        end
        sync()
      end
      $ 1628 "Direction: Base Z-"
      global move_thread_flag_1628=0
      thread move_thread_1628():
        enter_critical
        move_thread_flag_1628 = 1
        local towardsPos=calculate_point_to_move_towards(p[0.0,0.0,0.0,0.0,0.0,0.0], [0.0,0.0,-1.0], 1000.0)
        movel(towardsPos, a=0.007, v=0.007)
        move_thread_flag_1628 = 2
        exit_critical
      end
      move_thread_flag_1628 = 0
      move_thread_han_1628 = run move_thread_1628()
      while (True):
        local targetTcpDirection=get_target_tcp_speed()
        local stepsToRetract=tool_contact(direction=targetTcpDirection)
        if (stepsToRetract > 0):
          kill move_thread_han_1628
          stopl(0.02)
          local backTrackMovement=get_actual_joint_positions_history(stepsToRetract)
          local contactPose=get_forward_kin(backTrackMovement)
          local posDir=[targetTcpDirection[0],targetTcpDirection[1],targetTcpDirection[2]]
          local retractTo=contactPose
          if (norm(posDir) > 1e-6):
            local normalizedPosDir=normalize(posDir)
            local additionalRetraction=p[normalizedPosDir[0] * 0.0, normalizedPosDir[1] * 0.0, normalizedPosDir[2] * 0.0, 0, 0, 0]
            retractTo = pose_sub(contactPose, additionalRetraction)
          end
          movel(retractTo, a=0.02, v=0.1)
          $ 1629 "Until (tool_contact_detection)"
          break
        end
        sync()
      end
      $ 1630 "Popup: punto contacto alanzdo"
      popup("punto contacto alanzdo", "Mensaje", False, False, blocking=True)
      $ 1631 "Direction: Base Z+"
      global move_thread_flag_1631=0
      thread move_thread_1631():
        enter_critical
        move_thread_flag_1631 = 1
        local towardsPos=calculate_point_to_move_towards(p[0.0,0.0,0.0,0.0,0.0,0.0], [0.0,0.0,1.0], 0.002)
        movel(towardsPos, a=0.005, v=0.003)
        move_thread_flag_1631 = 2
        exit_critical
      end
      move_thread_flag_1631 = 0
      move_thread_han_1631 = run move_thread_1631()
      while (True):
        sleep(1.0E-10)
        if (move_thread_flag_1631 > 1):
          join move_thread_han_1631
          $ 1632 "Until (distance)"
          break
        end
        sync()
      end
      $ 1633 "Wait: 0.3"
      sleep(0.3)
      $ 1634 "Set CO[1]=Encender"
      set_configurable_digital_out(1, True)
      $ 1635 "Wait: 0.3"
      sleep(0.3)
      $ 1636 "Loop 1 times"
      Loop_129 = 0
      while (Loop_129 < 1):
        $ 1637 "bajar≔pose_add(get_actual_tcp_pose(), bajada_broca)"
        global bajar= pose_add ( get_actual_tcp_pose (), bajada_broca)
        $ 1638 "bajar" "breakAfter"
        movel(bajar, a=0.004, v=0.004)
        $ 1639 "subir≔pose_sub(get_actual_tcp_pose(), bajada_broca)"
        global subir= pose_sub ( get_actual_tcp_pose (), bajada_broca)
        $ 1640 "Direction: Base Z+"
        global move_thread_flag_1640=0
        thread move_thread_1640():
          enter_critical
          move_thread_flag_1640 = 1
          local towardsPos=calculate_point_to_move_towards(p[0.0,0.0,0.0,0.0,0.0,0.0], [0.0,0.0,1.0], 0.002)
          movel(towardsPos, a=0.015, v=0.015)
          move_thread_flag_1640 = 2
          exit_critical
        end
        move_thread_flag_1640 = 0
        move_thread_han_1640 = run move_thread_1640()
        while (True):
          sleep(1.0E-10)
          if (move_thread_flag_1640 > 1):
            join move_thread_han_1640
            $ 1641 "Until (distance)"
            break
          end
          sync()
        end
        $ 1642 "Set CO[1]=Apagar"
        set_configurable_digital_out(1, False)
        $ 1643 "subir" "breakAfter"
        movel(subir, a=0.015, v=0.015)
        $ 1644 "bajada_broca≔pose_sub(bajada_broca, bajada)"
        global bajada_broca= pose_sub (bajada_broca, bajada)
        Loop_129 = Loop_129 + 1
      end
      $ 1645 "Direction: Base Z+"
      global move_thread_flag_1645=0
      thread move_thread_1645():
        enter_critical
        move_thread_flag_1645 = 1
        local towardsPos=calculate_point_to_move_towards(p[0.0,0.0,0.0,0.0,0.0,0.0], [0.0,0.0,1.0], 0.08)
        movel(towardsPos, a=0.15, v=0.1)
        move_thread_flag_1645 = 2
        exit_critical
      end
      move_thread_flag_1645 = 0
      move_thread_han_1645 = run move_thread_1645()
      while (True):
        sleep(1.0E-10)
        if (move_thread_flag_1645 > 1):
          join move_thread_han_1645
          $ 1646 "Until (distance)"
          break
        end
        sync()
      end
      $ 1647 "Set CO[1]=Apagar"
      set_configurable_digital_out(1, False)
      $ 1648 "barreno_actual≔barreno_actual+1"
      global barreno_actual=barreno_actual+1
    end
    $ 1651 "Popup: Linea13 con chica Terminada!"
    popup("Linea13 con chica Terminada!", "Mensaje", False, False, blocking=True)
    $ 1652 "Linea14"
    $ 1653 "Marcar_puntos"
    $ 1654 "MoveL"
    $ 1655 "Linea14_A" "breakAfter"
    movel(Linea14_A_p, a=0.5, v=0.1)
    $ 1656 "bajada_comprobacion"
    $ 1657 "Direction: Base Z-"
    global move_thread_flag_1657=0
    thread move_thread_1657():
      enter_critical
      move_thread_flag_1657 = 1
      local towardsPos=calculate_point_to_move_towards(p[0.0,0.0,0.0,0.0,0.0,0.0], [0.0,0.0,-1.0], 0.071)
      movel(towardsPos, a=0.15, v=0.1)
      move_thread_flag_1657 = 2
      exit_critical
    end
    move_thread_flag_1657 = 0
    move_thread_han_1657 = run move_thread_1657()
    while (True):
      sleep(1.0E-10)
      if (move_thread_flag_1657 > 1):
        join move_thread_han_1657
        $ 1658 "Until (distance)"
        break
      end
      sync()
    end
    $ 1659 "Direction: Base Z-"
    global move_thread_flag_1659=0
    thread move_thread_1659():
      enter_critical
      move_thread_flag_1659 = 1
      local towardsPos=calculate_point_to_move_towards(p[0.0,0.0,0.0,0.0,0.0,0.0], [0.0,0.0,-1.0], 1000.0)
      movel(towardsPos, a=0.007, v=0.007)
      move_thread_flag_1659 = 2
      exit_critical
    end
    move_thread_flag_1659 = 0
    move_thread_han_1659 = run move_thread_1659()
    while (True):
      local targetTcpDirection=get_target_tcp_speed()
      local stepsToRetract=tool_contact(direction=targetTcpDirection)
      if (stepsToRetract > 0):
        kill move_thread_han_1659
        stopl(0.02)
        local backTrackMovement=get_actual_joint_positions_history(stepsToRetract)
        local contactPose=get_forward_kin(backTrackMovement)
        local posDir=[targetTcpDirection[0],targetTcpDirection[1],targetTcpDirection[2]]
        local retractTo=contactPose
        if (norm(posDir) > 1e-6):
          local normalizedPosDir=normalize(posDir)
          local additionalRetraction=p[normalizedPosDir[0] * 0.0, normalizedPosDir[1] * 0.0, normalizedPosDir[2] * 0.0, 0, 0, 0]
          retractTo = pose_sub(contactPose, additionalRetraction)
        end
        movel(retractTo, a=0.02, v=0.1)
        $ 1660 "Until (tool_contact_detection)"
        break
      end
      sync()
    end
    $ 1661 "Direction: Base Z+"
    global move_thread_flag_1661=0
    thread move_thread_1661():
      enter_critical
      move_thread_flag_1661 = 1
      local towardsPos=calculate_point_to_move_towards(p[0.0,0.0,0.0,0.0,0.0,0.0], [0.0,0.0,1.0], 0.08)
      movel(towardsPos, a=0.15, v=0.1)
      move_thread_flag_1661 = 2
      exit_critical
    end
    move_thread_flag_1661 = 0
    move_thread_han_1661 = run move_thread_1661()
    while (True):
      sleep(1.0E-10)
      if (move_thread_flag_1661 > 1):
        join move_thread_han_1661
        $ 1662 "Until (distance)"
        break
      end
      sync()
    end
    $ 1663 "Linea14_B" "breakAfter"
    movel(Linea14_B_p, a=0.5, v=0.1)
    $ 1664 "bajada_comprobacion"
    $ 1665 "Direction: Base Z-"
    global move_thread_flag_1665=0
    thread move_thread_1665():
      enter_critical
      move_thread_flag_1665 = 1
      local towardsPos=calculate_point_to_move_towards(p[0.0,0.0,0.0,0.0,0.0,0.0], [0.0,0.0,-1.0], 0.071)
      movel(towardsPos, a=0.15, v=0.1)
      move_thread_flag_1665 = 2
      exit_critical
    end
    move_thread_flag_1665 = 0
    move_thread_han_1665 = run move_thread_1665()
    while (True):
      sleep(1.0E-10)
      if (move_thread_flag_1665 > 1):
        join move_thread_han_1665
        $ 1666 "Until (distance)"
        break
      end
      sync()
    end
    $ 1667 "Direction: Base Z-"
    global move_thread_flag_1667=0
    thread move_thread_1667():
      enter_critical
      move_thread_flag_1667 = 1
      local towardsPos=calculate_point_to_move_towards(p[0.0,0.0,0.0,0.0,0.0,0.0], [0.0,0.0,-1.0], 1000.0)
      movel(towardsPos, a=0.007, v=0.007)
      move_thread_flag_1667 = 2
      exit_critical
    end
    move_thread_flag_1667 = 0
    move_thread_han_1667 = run move_thread_1667()
    while (True):
      local targetTcpDirection=get_target_tcp_speed()
      local stepsToRetract=tool_contact(direction=targetTcpDirection)
      if (stepsToRetract > 0):
        kill move_thread_han_1667
        stopl(0.02)
        local backTrackMovement=get_actual_joint_positions_history(stepsToRetract)
        local contactPose=get_forward_kin(backTrackMovement)
        local posDir=[targetTcpDirection[0],targetTcpDirection[1],targetTcpDirection[2]]
        local retractTo=contactPose
        if (norm(posDir) > 1e-6):
          local normalizedPosDir=normalize(posDir)
          local additionalRetraction=p[normalizedPosDir[0] * 0.0, normalizedPosDir[1] * 0.0, normalizedPosDir[2] * 0.0, 0, 0, 0]
          retractTo = pose_sub(contactPose, additionalRetraction)
        end
        movel(retractTo, a=0.02, v=0.1)
        $ 1668 "Until (tool_contact_detection)"
        break
      end
      sync()
    end
    $ 1669 "Direction: Base Z+"
    global move_thread_flag_1669=0
    thread move_thread_1669():
      enter_critical
      move_thread_flag_1669 = 1
      local towardsPos=calculate_point_to_move_towards(p[0.0,0.0,0.0,0.0,0.0,0.0], [0.0,0.0,1.0], 0.08)
      movel(towardsPos, a=0.15, v=0.1)
      move_thread_flag_1669 = 2
      exit_critical
    end
    move_thread_flag_1669 = 0
    move_thread_han_1669 = run move_thread_1669()
    while (True):
      sleep(1.0E-10)
      if (move_thread_flag_1669 > 1):
        join move_thread_han_1669
        $ 1670 "Until (distance)"
        break
      end
      sync()
    end
    $ 1671 "AB"
    $ 1672 "'desbaste_inicial'"
    # 'desbaste_inicial'
    $ 1673 "bajada_broca≔p[0,0,-0.008,0,0,0]"
    global bajada_broca=p[0,0,-0.008,0,0,0]
    $ 1674 "barrenos_menos1≔5"
    global barrenos_menos1=5
    $ 1675 "barreno_actual≔0"
    global barreno_actual=0
    $ 1676 "Loop barreno_actual≤barrenos_menos1"
    while (barreno_actual <= barrenos_menos1):
      $ 1677 "Perforacion"
      $ 1678 "MoveL"
      $ 1679 "If barreno_actual≟3"
      if (barreno_actual == 3):
        $ 1680 "barreno_actual≔barreno_actual+1"
        global barreno_actual=barreno_actual+1
      end
      $ 1681 "internos≔interpolate_pose(Linea14_A, Linea14_B, barreno_actual/barrenos_menos1)"
      global internos= interpolate_pose (Linea14_A_p, Linea14_B_p, barreno_actual/barrenos_menos1)
      $ 1682 "internos" "breakAfter"
      movel(internos, a=0.5, v=0.1)
      $ 1683 "'desbaste_inicial'"
      # 'desbaste_inicial'
      $ 1684 "bajada_broca≔p[0,0,-0.024,0,0,0]"
      global bajada_broca=p[0,0,-0.024,0,0,0]
      $ 1685 "bajada≔p[0,0,0.024,0,0,0]"
      global bajada=p[0,0,0.024,0,0,0]
      $ 1686 "Direction: Base Z-"
      global move_thread_flag_1686=0
      thread move_thread_1686():
        enter_critical
        move_thread_flag_1686 = 1
        local towardsPos=calculate_point_to_move_towards(p[0.0,0.0,0.0,0.0,0.0,0.0], [0.0,0.0,-1.0], 0.071)
        movel(towardsPos, a=0.15, v=0.1)
        move_thread_flag_1686 = 2
        exit_critical
      end
      move_thread_flag_1686 = 0
      move_thread_han_1686 = run move_thread_1686()
      while (True):
        sleep(1.0E-10)
        if (move_thread_flag_1686 > 1):
          join move_thread_han_1686
          $ 1687 "Until (distance)"
          break
        end
        sync()
      end
      $ 1688 "Direction: Base Z-"
      global move_thread_flag_1688=0
      thread move_thread_1688():
        enter_critical
        move_thread_flag_1688 = 1
        local towardsPos=calculate_point_to_move_towards(p[0.0,0.0,0.0,0.0,0.0,0.0], [0.0,0.0,-1.0], 1000.0)
        movel(towardsPos, a=0.007, v=0.007)
        move_thread_flag_1688 = 2
        exit_critical
      end
      move_thread_flag_1688 = 0
      move_thread_han_1688 = run move_thread_1688()
      while (True):
        local targetTcpDirection=get_target_tcp_speed()
        local stepsToRetract=tool_contact(direction=targetTcpDirection)
        if (stepsToRetract > 0):
          kill move_thread_han_1688
          stopl(0.02)
          local backTrackMovement=get_actual_joint_positions_history(stepsToRetract)
          local contactPose=get_forward_kin(backTrackMovement)
          local posDir=[targetTcpDirection[0],targetTcpDirection[1],targetTcpDirection[2]]
          local retractTo=contactPose
          if (norm(posDir) > 1e-6):
            local normalizedPosDir=normalize(posDir)
            local additionalRetraction=p[normalizedPosDir[0] * 0.0, normalizedPosDir[1] * 0.0, normalizedPosDir[2] * 0.0, 0, 0, 0]
            retractTo = pose_sub(contactPose, additionalRetraction)
          end
          movel(retractTo, a=0.02, v=0.1)
          $ 1689 "Until (tool_contact_detection)"
          break
        end
        sync()
      end
      $ 1690 "Popup: punto contacto alanzdo"
      popup("punto contacto alanzdo", "Mensaje", False, False, blocking=True)
      $ 1691 "Direction: Base Z+"
      global move_thread_flag_1691=0
      thread move_thread_1691():
        enter_critical
        move_thread_flag_1691 = 1
        local towardsPos=calculate_point_to_move_towards(p[0.0,0.0,0.0,0.0,0.0,0.0], [0.0,0.0,1.0], 0.002)
        movel(towardsPos, a=0.005, v=0.003)
        move_thread_flag_1691 = 2
        exit_critical
      end
      move_thread_flag_1691 = 0
      move_thread_han_1691 = run move_thread_1691()
      while (True):
        sleep(1.0E-10)
        if (move_thread_flag_1691 > 1):
          join move_thread_han_1691
          $ 1692 "Until (distance)"
          break
        end
        sync()
      end
      $ 1693 "Wait: 0.3"
      sleep(0.3)
      $ 1694 "Set CO[1]=Encender"
      set_configurable_digital_out(1, True)
      $ 1695 "Wait: 0.3"
      sleep(0.3)
      $ 1696 "Loop 1 times"
      Loop_131 = 0
      while (Loop_131 < 1):
        $ 1697 "bajar≔pose_add(get_actual_tcp_pose(), bajada_broca)"
        global bajar= pose_add ( get_actual_tcp_pose (), bajada_broca)
        $ 1698 "bajar" "breakAfter"
        movel(bajar, a=0.004, v=0.004)
        $ 1699 "subir≔pose_sub(get_actual_tcp_pose(), bajada_broca)"
        global subir= pose_sub ( get_actual_tcp_pose (), bajada_broca)
        $ 1700 "Direction: Base Z+"
        global move_thread_flag_1700=0
        thread move_thread_1700():
          enter_critical
          move_thread_flag_1700 = 1
          local towardsPos=calculate_point_to_move_towards(p[0.0,0.0,0.0,0.0,0.0,0.0], [0.0,0.0,1.0], 0.002)
          movel(towardsPos, a=0.015, v=0.015)
          move_thread_flag_1700 = 2
          exit_critical
        end
        move_thread_flag_1700 = 0
        move_thread_han_1700 = run move_thread_1700()
        while (True):
          sleep(1.0E-10)
          if (move_thread_flag_1700 > 1):
            join move_thread_han_1700
            $ 1701 "Until (distance)"
            break
          end
          sync()
        end
        $ 1702 "Set CO[1]=Apagar"
        set_configurable_digital_out(1, False)
        $ 1703 "subir" "breakAfter"
        movel(subir, a=0.015, v=0.015)
        $ 1704 "bajada_broca≔pose_sub(bajada_broca, bajada)"
        global bajada_broca= pose_sub (bajada_broca, bajada)
        Loop_131 = Loop_131 + 1
      end
      $ 1705 "Direction: Base Z+"
      global move_thread_flag_1705=0
      thread move_thread_1705():
        enter_critical
        move_thread_flag_1705 = 1
        local towardsPos=calculate_point_to_move_towards(p[0.0,0.0,0.0,0.0,0.0,0.0], [0.0,0.0,1.0], 0.08)
        movel(towardsPos, a=0.15, v=0.1)
        move_thread_flag_1705 = 2
        exit_critical
      end
      move_thread_flag_1705 = 0
      move_thread_han_1705 = run move_thread_1705()
      while (True):
        sleep(1.0E-10)
        if (move_thread_flag_1705 > 1):
          join move_thread_han_1705
          $ 1706 "Until (distance)"
          break
        end
        sync()
      end
      $ 1707 "Set CO[1]=Apagar"
      set_configurable_digital_out(1, False)
      $ 1708 "barreno_actual≔barreno_actual+1"
      global barreno_actual=barreno_actual+1
    end
    $ 1711 "Popup: Linea14 con chica Terminada!"
    popup("Linea14 con chica Terminada!", "Mensaje", False, False, blocking=True)
    $ 1712 "Linea15"
    $ 1713 "Marcar_puntos"
    $ 1714 "MoveL"
    $ 1715 "Linea15_A" "breakAfter"
    movel(Linea15_A_p, a=0.5, v=0.1)
    $ 1716 "bajada_comprobacion"
    $ 1717 "Direction: Base Z-"
    global move_thread_flag_1717=0
    thread move_thread_1717():
      enter_critical
      move_thread_flag_1717 = 1
      local towardsPos=calculate_point_to_move_towards(p[0.0,0.0,0.0,0.0,0.0,0.0], [0.0,0.0,-1.0], 0.071)
      movel(towardsPos, a=0.15, v=0.1)
      move_thread_flag_1717 = 2
      exit_critical
    end
    move_thread_flag_1717 = 0
    move_thread_han_1717 = run move_thread_1717()
    while (True):
      sleep(1.0E-10)
      if (move_thread_flag_1717 > 1):
        join move_thread_han_1717
        $ 1718 "Until (distance)"
        break
      end
      sync()
    end
    $ 1719 "Direction: Base Z-"
    global move_thread_flag_1719=0
    thread move_thread_1719():
      enter_critical
      move_thread_flag_1719 = 1
      local towardsPos=calculate_point_to_move_towards(p[0.0,0.0,0.0,0.0,0.0,0.0], [0.0,0.0,-1.0], 1000.0)
      movel(towardsPos, a=0.007, v=0.007)
      move_thread_flag_1719 = 2
      exit_critical
    end
    move_thread_flag_1719 = 0
    move_thread_han_1719 = run move_thread_1719()
    while (True):
      local targetTcpDirection=get_target_tcp_speed()
      local stepsToRetract=tool_contact(direction=targetTcpDirection)
      if (stepsToRetract > 0):
        kill move_thread_han_1719
        stopl(0.02)
        local backTrackMovement=get_actual_joint_positions_history(stepsToRetract)
        local contactPose=get_forward_kin(backTrackMovement)
        local posDir=[targetTcpDirection[0],targetTcpDirection[1],targetTcpDirection[2]]
        local retractTo=contactPose
        if (norm(posDir) > 1e-6):
          local normalizedPosDir=normalize(posDir)
          local additionalRetraction=p[normalizedPosDir[0] * 0.0, normalizedPosDir[1] * 0.0, normalizedPosDir[2] * 0.0, 0, 0, 0]
          retractTo = pose_sub(contactPose, additionalRetraction)
        end
        movel(retractTo, a=0.02, v=0.1)
        $ 1720 "Until (tool_contact_detection)"
        break
      end
      sync()
    end
    $ 1721 "Direction: Base Z+"
    global move_thread_flag_1721=0
    thread move_thread_1721():
      enter_critical
      move_thread_flag_1721 = 1
      local towardsPos=calculate_point_to_move_towards(p[0.0,0.0,0.0,0.0,0.0,0.0], [0.0,0.0,1.0], 0.08)
      movel(towardsPos, a=0.15, v=0.1)
      move_thread_flag_1721 = 2
      exit_critical
    end
    move_thread_flag_1721 = 0
    move_thread_han_1721 = run move_thread_1721()
    while (True):
      sleep(1.0E-10)
      if (move_thread_flag_1721 > 1):
        join move_thread_han_1721
        $ 1722 "Until (distance)"
        break
      end
      sync()
    end
    $ 1723 "Linea15_B" "breakAfter"
    movel(Linea15_B_p, a=0.5, v=0.1)
    $ 1724 "bajada_comprobacion"
    $ 1725 "Direction: Base Z-"
    global move_thread_flag_1725=0
    thread move_thread_1725():
      enter_critical
      move_thread_flag_1725 = 1
      local towardsPos=calculate_point_to_move_towards(p[0.0,0.0,0.0,0.0,0.0,0.0], [0.0,0.0,-1.0], 0.071)
      movel(towardsPos, a=0.15, v=0.1)
      move_thread_flag_1725 = 2
      exit_critical
    end
    move_thread_flag_1725 = 0
    move_thread_han_1725 = run move_thread_1725()
    while (True):
      sleep(1.0E-10)
      if (move_thread_flag_1725 > 1):
        join move_thread_han_1725
        $ 1726 "Until (distance)"
        break
      end
      sync()
    end
    $ 1727 "Direction: Base Z-"
    global move_thread_flag_1727=0
    thread move_thread_1727():
      enter_critical
      move_thread_flag_1727 = 1
      local towardsPos=calculate_point_to_move_towards(p[0.0,0.0,0.0,0.0,0.0,0.0], [0.0,0.0,-1.0], 1000.0)
      movel(towardsPos, a=0.007, v=0.007)
      move_thread_flag_1727 = 2
      exit_critical
    end
    move_thread_flag_1727 = 0
    move_thread_han_1727 = run move_thread_1727()
    while (True):
      local targetTcpDirection=get_target_tcp_speed()
      local stepsToRetract=tool_contact(direction=targetTcpDirection)
      if (stepsToRetract > 0):
        kill move_thread_han_1727
        stopl(0.02)
        local backTrackMovement=get_actual_joint_positions_history(stepsToRetract)
        local contactPose=get_forward_kin(backTrackMovement)
        local posDir=[targetTcpDirection[0],targetTcpDirection[1],targetTcpDirection[2]]
        local retractTo=contactPose
        if (norm(posDir) > 1e-6):
          local normalizedPosDir=normalize(posDir)
          local additionalRetraction=p[normalizedPosDir[0] * 0.0, normalizedPosDir[1] * 0.0, normalizedPosDir[2] * 0.0, 0, 0, 0]
          retractTo = pose_sub(contactPose, additionalRetraction)
        end
        movel(retractTo, a=0.02, v=0.1)
        $ 1728 "Until (tool_contact_detection)"
        break
      end
      sync()
    end
    $ 1729 "Direction: Base Z+"
    global move_thread_flag_1729=0
    thread move_thread_1729():
      enter_critical
      move_thread_flag_1729 = 1
      local towardsPos=calculate_point_to_move_towards(p[0.0,0.0,0.0,0.0,0.0,0.0], [0.0,0.0,1.0], 0.08)
      movel(towardsPos, a=0.15, v=0.1)
      move_thread_flag_1729 = 2
      exit_critical
    end
    move_thread_flag_1729 = 0
    move_thread_han_1729 = run move_thread_1729()
    while (True):
      sleep(1.0E-10)
      if (move_thread_flag_1729 > 1):
        join move_thread_han_1729
        $ 1730 "Until (distance)"
        break
      end
      sync()
    end
    $ 1731 "AB"
    $ 1732 "'desbaste_inicial'"
    # 'desbaste_inicial'
    $ 1733 "bajada_broca≔p[0,0,-0.008,0,0,0]"
    global bajada_broca=p[0,0,-0.008,0,0,0]
    $ 1734 "barrenos_menos1≔3"
    global barrenos_menos1=3
    $ 1735 "barreno_actual≔0"
    global barreno_actual=0
    $ 1736 "Loop barreno_actual≤barrenos_menos1"
    while (barreno_actual <= barrenos_menos1):
      $ 1737 "Perforacion"
      $ 1738 "MoveL"
      $ 1741 "internos≔interpolate_pose(Linea15_A, Linea15_B, barreno_actual/barrenos_menos1)"
      global internos= interpolate_pose (Linea15_A_p, Linea15_B_p, barreno_actual/barrenos_menos1)
      $ 1742 "internos" "breakAfter"
      movel(internos, a=0.5, v=0.1)
      $ 1743 "'desbaste_inicial'"
      # 'desbaste_inicial'
      $ 1744 "bajada_broca≔p[0,0,-0.024,0,0,0]"
      global bajada_broca=p[0,0,-0.024,0,0,0]
      $ 1745 "bajada≔p[0,0,0.024,0,0,0]"
      global bajada=p[0,0,0.024,0,0,0]
      $ 1746 "Direction: Base Z-"
      global move_thread_flag_1746=0
      thread move_thread_1746():
        enter_critical
        move_thread_flag_1746 = 1
        local towardsPos=calculate_point_to_move_towards(p[0.0,0.0,0.0,0.0,0.0,0.0], [0.0,0.0,-1.0], 0.071)
        movel(towardsPos, a=0.15, v=0.1)
        move_thread_flag_1746 = 2
        exit_critical
      end
      move_thread_flag_1746 = 0
      move_thread_han_1746 = run move_thread_1746()
      while (True):
        sleep(1.0E-10)
        if (move_thread_flag_1746 > 1):
          join move_thread_han_1746
          $ 1747 "Until (distance)"
          break
        end
        sync()
      end
      $ 1748 "Direction: Base Z-"
      global move_thread_flag_1748=0
      thread move_thread_1748():
        enter_critical
        move_thread_flag_1748 = 1
        local towardsPos=calculate_point_to_move_towards(p[0.0,0.0,0.0,0.0,0.0,0.0], [0.0,0.0,-1.0], 1000.0)
        movel(towardsPos, a=0.007, v=0.007)
        move_thread_flag_1748 = 2
        exit_critical
      end
      move_thread_flag_1748 = 0
      move_thread_han_1748 = run move_thread_1748()
      while (True):
        local targetTcpDirection=get_target_tcp_speed()
        local stepsToRetract=tool_contact(direction=targetTcpDirection)
        if (stepsToRetract > 0):
          kill move_thread_han_1748
          stopl(0.02)
          local backTrackMovement=get_actual_joint_positions_history(stepsToRetract)
          local contactPose=get_forward_kin(backTrackMovement)
          local posDir=[targetTcpDirection[0],targetTcpDirection[1],targetTcpDirection[2]]
          local retractTo=contactPose
          if (norm(posDir) > 1e-6):
            local normalizedPosDir=normalize(posDir)
            local additionalRetraction=p[normalizedPosDir[0] * 0.0, normalizedPosDir[1] * 0.0, normalizedPosDir[2] * 0.0, 0, 0, 0]
            retractTo = pose_sub(contactPose, additionalRetraction)
          end
          movel(retractTo, a=0.02, v=0.1)
          $ 1749 "Until (tool_contact_detection)"
          break
        end
        sync()
      end
      $ 1750 "Popup: punto contacto alanzdo"
      popup("punto contacto alanzdo", "Mensaje", False, False, blocking=True)
      $ 1751 "Direction: Base Z+"
      global move_thread_flag_1751=0
      thread move_thread_1751():
        enter_critical
        move_thread_flag_1751 = 1
        local towardsPos=calculate_point_to_move_towards(p[0.0,0.0,0.0,0.0,0.0,0.0], [0.0,0.0,1.0], 0.002)
        movel(towardsPos, a=0.005, v=0.003)
        move_thread_flag_1751 = 2
        exit_critical
      end
      move_thread_flag_1751 = 0
      move_thread_han_1751 = run move_thread_1751()
      while (True):
        sleep(1.0E-10)
        if (move_thread_flag_1751 > 1):
          join move_thread_han_1751
          $ 1752 "Until (distance)"
          break
        end
        sync()
      end
      $ 1753 "Wait: 0.3"
      sleep(0.3)
      $ 1754 "Set CO[1]=Encender"
      set_configurable_digital_out(1, True)
      $ 1755 "Wait: 0.3"
      sleep(0.3)
      $ 1756 "Loop 1 times"
      Loop_133 = 0
      while (Loop_133 < 1):
        $ 1757 "bajar≔pose_add(get_actual_tcp_pose(), bajada_broca)"
        global bajar= pose_add ( get_actual_tcp_pose (), bajada_broca)
        $ 1758 "bajar" "breakAfter"
        movel(bajar, a=0.004, v=0.004)
        $ 1759 "subir≔pose_sub(get_actual_tcp_pose(), bajada_broca)"
        global subir= pose_sub ( get_actual_tcp_pose (), bajada_broca)
        $ 1760 "Direction: Base Z+"
        global move_thread_flag_1760=0
        thread move_thread_1760():
          enter_critical
          move_thread_flag_1760 = 1
          local towardsPos=calculate_point_to_move_towards(p[0.0,0.0,0.0,0.0,0.0,0.0], [0.0,0.0,1.0], 0.002)
          movel(towardsPos, a=0.015, v=0.015)
          move_thread_flag_1760 = 2
          exit_critical
        end
        move_thread_flag_1760 = 0
        move_thread_han_1760 = run move_thread_1760()
        while (True):
          sleep(1.0E-10)
          if (move_thread_flag_1760 > 1):
            join move_thread_han_1760
            $ 1761 "Until (distance)"
            break
          end
          sync()
        end
        $ 1762 "Set CO[1]=Apagar"
        set_configurable_digital_out(1, False)
        $ 1763 "subir" "breakAfter"
        movel(subir, a=0.015, v=0.015)
        $ 1764 "bajada_broca≔pose_sub(bajada_broca, bajada)"
        global bajada_broca= pose_sub (bajada_broca, bajada)
        Loop_133 = Loop_133 + 1
      end
      $ 1765 "Direction: Base Z+"
      global move_thread_flag_1765=0
      thread move_thread_1765():
        enter_critical
        move_thread_flag_1765 = 1
        local towardsPos=calculate_point_to_move_towards(p[0.0,0.0,0.0,0.0,0.0,0.0], [0.0,0.0,1.0], 0.08)
        movel(towardsPos, a=0.15, v=0.1)
        move_thread_flag_1765 = 2
        exit_critical
      end
      move_thread_flag_1765 = 0
      move_thread_han_1765 = run move_thread_1765()
      while (True):
        sleep(1.0E-10)
        if (move_thread_flag_1765 > 1):
          join move_thread_han_1765
          $ 1766 "Until (distance)"
          break
        end
        sync()
      end
      $ 1767 "Set CO[1]=Apagar"
      set_configurable_digital_out(1, False)
      $ 1768 "barreno_actual≔barreno_actual+1"
      global barreno_actual=barreno_actual+1
    end
    $ 1771 "Popup: Linea15 con chica Terminada!"
    popup("Linea15 con chica Terminada!", "Mensaje", False, False, blocking=True)
    $ 1772 "Linea16"
    $ 1773 "Marcar_puntos"
    $ 1774 "MoveL"
    $ 1775 "Linea16_A" "breakAfter"
    movel(Linea16_A_p, a=0.5, v=0.1)
    $ 1776 "bajada_comprobacion"
    $ 1777 "Direction: Base Z-"
    global move_thread_flag_1777=0
    thread move_thread_1777():
      enter_critical
      move_thread_flag_1777 = 1
      local towardsPos=calculate_point_to_move_towards(p[0.0,0.0,0.0,0.0,0.0,0.0], [0.0,0.0,-1.0], 0.071)
      movel(towardsPos, a=0.15, v=0.1)
      move_thread_flag_1777 = 2
      exit_critical
    end
    move_thread_flag_1777 = 0
    move_thread_han_1777 = run move_thread_1777()
    while (True):
      sleep(1.0E-10)
      if (move_thread_flag_1777 > 1):
        join move_thread_han_1777
        $ 1778 "Until (distance)"
        break
      end
      sync()
    end
    $ 1779 "Direction: Base Z-"
    global move_thread_flag_1779=0
    thread move_thread_1779():
      enter_critical
      move_thread_flag_1779 = 1
      local towardsPos=calculate_point_to_move_towards(p[0.0,0.0,0.0,0.0,0.0,0.0], [0.0,0.0,-1.0], 1000.0)
      movel(towardsPos, a=0.007, v=0.007)
      move_thread_flag_1779 = 2
      exit_critical
    end
    move_thread_flag_1779 = 0
    move_thread_han_1779 = run move_thread_1779()
    while (True):
      local targetTcpDirection=get_target_tcp_speed()
      local stepsToRetract=tool_contact(direction=targetTcpDirection)
      if (stepsToRetract > 0):
        kill move_thread_han_1779
        stopl(0.02)
        local backTrackMovement=get_actual_joint_positions_history(stepsToRetract)
        local contactPose=get_forward_kin(backTrackMovement)
        local posDir=[targetTcpDirection[0],targetTcpDirection[1],targetTcpDirection[2]]
        local retractTo=contactPose
        if (norm(posDir) > 1e-6):
          local normalizedPosDir=normalize(posDir)
          local additionalRetraction=p[normalizedPosDir[0] * 0.0, normalizedPosDir[1] * 0.0, normalizedPosDir[2] * 0.0, 0, 0, 0]
          retractTo = pose_sub(contactPose, additionalRetraction)
        end
        movel(retractTo, a=0.02, v=0.1)
        $ 1780 "Until (tool_contact_detection)"
        break
      end
      sync()
    end
    $ 1781 "Direction: Base Z+"
    global move_thread_flag_1781=0
    thread move_thread_1781():
      enter_critical
      move_thread_flag_1781 = 1
      local towardsPos=calculate_point_to_move_towards(p[0.0,0.0,0.0,0.0,0.0,0.0], [0.0,0.0,1.0], 0.08)
      movel(towardsPos, a=0.15, v=0.1)
      move_thread_flag_1781 = 2
      exit_critical
    end
    move_thread_flag_1781 = 0
    move_thread_han_1781 = run move_thread_1781()
    while (True):
      sleep(1.0E-10)
      if (move_thread_flag_1781 > 1):
        join move_thread_han_1781
        $ 1782 "Until (distance)"
        break
      end
      sync()
    end
    $ 1783 "Linea16_B" "breakAfter"
    movel(Linea16_B_p, a=0.5, v=0.1)
    $ 1784 "bajada_comprobacion"
    $ 1785 "Direction: Base Z-"
    global move_thread_flag_1785=0
    thread move_thread_1785():
      enter_critical
      move_thread_flag_1785 = 1
      local towardsPos=calculate_point_to_move_towards(p[0.0,0.0,0.0,0.0,0.0,0.0], [0.0,0.0,-1.0], 0.071)
      movel(towardsPos, a=0.15, v=0.1)
      move_thread_flag_1785 = 2
      exit_critical
    end
    move_thread_flag_1785 = 0
    move_thread_han_1785 = run move_thread_1785()
    while (True):
      sleep(1.0E-10)
      if (move_thread_flag_1785 > 1):
        join move_thread_han_1785
        $ 1786 "Until (distance)"
        break
      end
      sync()
    end
    $ 1787 "Direction: Base Z-"
    global move_thread_flag_1787=0
    thread move_thread_1787():
      enter_critical
      move_thread_flag_1787 = 1
      local towardsPos=calculate_point_to_move_towards(p[0.0,0.0,0.0,0.0,0.0,0.0], [0.0,0.0,-1.0], 1000.0)
      movel(towardsPos, a=0.007, v=0.007)
      move_thread_flag_1787 = 2
      exit_critical
    end
    move_thread_flag_1787 = 0
    move_thread_han_1787 = run move_thread_1787()
    while (True):
      local targetTcpDirection=get_target_tcp_speed()
      local stepsToRetract=tool_contact(direction=targetTcpDirection)
      if (stepsToRetract > 0):
        kill move_thread_han_1787
        stopl(0.02)
        local backTrackMovement=get_actual_joint_positions_history(stepsToRetract)
        local contactPose=get_forward_kin(backTrackMovement)
        local posDir=[targetTcpDirection[0],targetTcpDirection[1],targetTcpDirection[2]]
        local retractTo=contactPose
        if (norm(posDir) > 1e-6):
          local normalizedPosDir=normalize(posDir)
          local additionalRetraction=p[normalizedPosDir[0] * 0.0, normalizedPosDir[1] * 0.0, normalizedPosDir[2] * 0.0, 0, 0, 0]
          retractTo = pose_sub(contactPose, additionalRetraction)
        end
        movel(retractTo, a=0.02, v=0.1)
        $ 1788 "Until (tool_contact_detection)"
        break
      end
      sync()
    end
    $ 1789 "Direction: Base Z+"
    global move_thread_flag_1789=0
    thread move_thread_1789():
      enter_critical
      move_thread_flag_1789 = 1
      local towardsPos=calculate_point_to_move_towards(p[0.0,0.0,0.0,0.0,0.0,0.0], [0.0,0.0,1.0], 0.08)
      movel(towardsPos, a=0.15, v=0.1)
      move_thread_flag_1789 = 2
      exit_critical
    end
    move_thread_flag_1789 = 0
    move_thread_han_1789 = run move_thread_1789()
    while (True):
      sleep(1.0E-10)
      if (move_thread_flag_1789 > 1):
        join move_thread_han_1789
        $ 1790 "Until (distance)"
        break
      end
      sync()
    end
    $ 1791 "AB"
    $ 1792 "'desbaste_inicial'"
    # 'desbaste_inicial'
    $ 1793 "bajada_broca≔p[0,0,-0.008,0,0,0]"
    global bajada_broca=p[0,0,-0.008,0,0,0]
    $ 1794 "barrenos_menos1≔1"
    global barrenos_menos1=1
    $ 1795 "barreno_actual≔0"
    global barreno_actual=0
    $ 1796 "Loop barreno_actual≤barrenos_menos1"
    while (barreno_actual <= barrenos_menos1):
      $ 1797 "Perforacion"
      $ 1798 "MoveL"
      $ 1801 "internos≔interpolate_pose(Linea16_A, Linea16_B, barreno_actual/barrenos_menos1)"
      global internos= interpolate_pose (Linea16_A_p, Linea16_B_p, barreno_actual/barrenos_menos1)
      $ 1802 "internos" "breakAfter"
      movel(internos, a=0.5, v=0.1)
      $ 1803 "'desbaste_inicial'"
      # 'desbaste_inicial'
      $ 1804 "bajada_broca≔p[0,0,-0.024,0,0,0]"
      global bajada_broca=p[0,0,-0.024,0,0,0]
      $ 1805 "bajada≔p[0,0,0.024,0,0,0]"
      global bajada=p[0,0,0.024,0,0,0]
      $ 1806 "Direction: Base Z-"
      global move_thread_flag_1806=0
      thread move_thread_1806():
        enter_critical
        move_thread_flag_1806 = 1
        local towardsPos=calculate_point_to_move_towards(p[0.0,0.0,0.0,0.0,0.0,0.0], [0.0,0.0,-1.0], 0.071)
        movel(towardsPos, a=0.15, v=0.1)
        move_thread_flag_1806 = 2
        exit_critical
      end
      move_thread_flag_1806 = 0
      move_thread_han_1806 = run move_thread_1806()
      while (True):
        sleep(1.0E-10)
        if (move_thread_flag_1806 > 1):
          join move_thread_han_1806
          $ 1807 "Until (distance)"
          break
        end
        sync()
      end
      $ 1808 "Direction: Base Z-"
      global move_thread_flag_1808=0
      thread move_thread_1808():
        enter_critical
        move_thread_flag_1808 = 1
        local towardsPos=calculate_point_to_move_towards(p[0.0,0.0,0.0,0.0,0.0,0.0], [0.0,0.0,-1.0], 1000.0)
        movel(towardsPos, a=0.007, v=0.007)
        move_thread_flag_1808 = 2
        exit_critical
      end
      move_thread_flag_1808 = 0
      move_thread_han_1808 = run move_thread_1808()
      while (True):
        local targetTcpDirection=get_target_tcp_speed()
        local stepsToRetract=tool_contact(direction=targetTcpDirection)
        if (stepsToRetract > 0):
          kill move_thread_han_1808
          stopl(0.02)
          local backTrackMovement=get_actual_joint_positions_history(stepsToRetract)
          local contactPose=get_forward_kin(backTrackMovement)
          local posDir=[targetTcpDirection[0],targetTcpDirection[1],targetTcpDirection[2]]
          local retractTo=contactPose
          if (norm(posDir) > 1e-6):
            local normalizedPosDir=normalize(posDir)
            local additionalRetraction=p[normalizedPosDir[0] * 0.0, normalizedPosDir[1] * 0.0, normalizedPosDir[2] * 0.0, 0, 0, 0]
            retractTo = pose_sub(contactPose, additionalRetraction)
          end
          movel(retractTo, a=0.02, v=0.1)
          $ 1809 "Until (tool_contact_detection)"
          break
        end
        sync()
      end
      $ 1810 "Popup: punto contacto alanzdo"
      popup("punto contacto alanzdo", "Mensaje", False, False, blocking=True)
      $ 1811 "Direction: Base Z+"
      global move_thread_flag_1811=0
      thread move_thread_1811():
        enter_critical
        move_thread_flag_1811 = 1
        local towardsPos=calculate_point_to_move_towards(p[0.0,0.0,0.0,0.0,0.0,0.0], [0.0,0.0,1.0], 0.002)
        movel(towardsPos, a=0.005, v=0.003)
        move_thread_flag_1811 = 2
        exit_critical
      end
      move_thread_flag_1811 = 0
      move_thread_han_1811 = run move_thread_1811()
      while (True):
        sleep(1.0E-10)
        if (move_thread_flag_1811 > 1):
          join move_thread_han_1811
          $ 1812 "Until (distance)"
          break
        end
        sync()
      end
      $ 1813 "Wait: 0.3"
      sleep(0.3)
      $ 1814 "Set CO[1]=Encender"
      set_configurable_digital_out(1, True)
      $ 1815 "Wait: 0.3"
      sleep(0.3)
      $ 1816 "Loop 1 times"
      Loop_135 = 0
      while (Loop_135 < 1):
        $ 1817 "bajar≔pose_add(get_actual_tcp_pose(), bajada_broca)"
        global bajar= pose_add ( get_actual_tcp_pose (), bajada_broca)
        $ 1818 "bajar" "breakAfter"
        movel(bajar, a=0.004, v=0.004)
        $ 1819 "subir≔pose_sub(get_actual_tcp_pose(), bajada_broca)"
        global subir= pose_sub ( get_actual_tcp_pose (), bajada_broca)
        $ 1820 "Direction: Base Z+"
        global move_thread_flag_1820=0
        thread move_thread_1820():
          enter_critical
          move_thread_flag_1820 = 1
          local towardsPos=calculate_point_to_move_towards(p[0.0,0.0,0.0,0.0,0.0,0.0], [0.0,0.0,1.0], 0.002)
          movel(towardsPos, a=0.015, v=0.015)
          move_thread_flag_1820 = 2
          exit_critical
        end
        move_thread_flag_1820 = 0
        move_thread_han_1820 = run move_thread_1820()
        while (True):
          sleep(1.0E-10)
          if (move_thread_flag_1820 > 1):
            join move_thread_han_1820
            $ 1821 "Until (distance)"
            break
          end
          sync()
        end
        $ 1822 "Set CO[1]=Apagar"
        set_configurable_digital_out(1, False)
        $ 1823 "subir" "breakAfter"
        movel(subir, a=0.015, v=0.015)
        $ 1824 "bajada_broca≔pose_sub(bajada_broca, bajada)"
        global bajada_broca= pose_sub (bajada_broca, bajada)
        Loop_135 = Loop_135 + 1
      end
      $ 1825 "Direction: Base Z+"
      global move_thread_flag_1825=0
      thread move_thread_1825():
        enter_critical
        move_thread_flag_1825 = 1
        local towardsPos=calculate_point_to_move_towards(p[0.0,0.0,0.0,0.0,0.0,0.0], [0.0,0.0,1.0], 0.08)
        movel(towardsPos, a=0.15, v=0.1)
        move_thread_flag_1825 = 2
        exit_critical
      end
      move_thread_flag_1825 = 0
      move_thread_han_1825 = run move_thread_1825()
      while (True):
        sleep(1.0E-10)
        if (move_thread_flag_1825 > 1):
          join move_thread_han_1825
          $ 1826 "Until (distance)"
          break
        end
        sync()
      end
      $ 1827 "Set CO[1]=Apagar"
      set_configurable_digital_out(1, False)
      $ 1828 "barreno_actual≔barreno_actual+1"
      global barreno_actual=barreno_actual+1
    end
    $ 1831 "Popup: Linea16 con chica Terminada!"
    popup("Linea16 con chica Terminada!", "Mensaje", False, False, blocking=True)
    $ 1832 "Linea17"
    $ 1833 "Marcar_puntos"
    $ 1834 "MoveL"
    $ 1835 "Linea17_A" "breakAfter"
    movel(Linea17_A_p, a=0.5, v=0.1)
    $ 1836 "bajada_comprobacion"
    $ 1837 "Direction: Base Z-"
    global move_thread_flag_1837=0
    thread move_thread_1837():
      enter_critical
      move_thread_flag_1837 = 1
      local towardsPos=calculate_point_to_move_towards(p[0.0,0.0,0.0,0.0,0.0,0.0], [0.0,0.0,-1.0], 0.071)
      movel(towardsPos, a=0.15, v=0.1)
      move_thread_flag_1837 = 2
      exit_critical
    end
    move_thread_flag_1837 = 0
    move_thread_han_1837 = run move_thread_1837()
    while (True):
      sleep(1.0E-10)
      if (move_thread_flag_1837 > 1):
        join move_thread_han_1837
        $ 1838 "Until (distance)"
        break
      end
      sync()
    end
    $ 1839 "Direction: Base Z-"
    global move_thread_flag_1839=0
    thread move_thread_1839():
      enter_critical
      move_thread_flag_1839 = 1
      local towardsPos=calculate_point_to_move_towards(p[0.0,0.0,0.0,0.0,0.0,0.0], [0.0,0.0,-1.0], 1000.0)
      movel(towardsPos, a=0.007, v=0.007)
      move_thread_flag_1839 = 2
      exit_critical
    end
    move_thread_flag_1839 = 0
    move_thread_han_1839 = run move_thread_1839()
    while (True):
      local targetTcpDirection=get_target_tcp_speed()
      local stepsToRetract=tool_contact(direction=targetTcpDirection)
      if (stepsToRetract > 0):
        kill move_thread_han_1839
        stopl(0.02)
        local backTrackMovement=get_actual_joint_positions_history(stepsToRetract)
        local contactPose=get_forward_kin(backTrackMovement)
        local posDir=[targetTcpDirection[0],targetTcpDirection[1],targetTcpDirection[2]]
        local retractTo=contactPose
        if (norm(posDir) > 1e-6):
          local normalizedPosDir=normalize(posDir)
          local additionalRetraction=p[normalizedPosDir[0] * 0.0, normalizedPosDir[1] * 0.0, normalizedPosDir[2] * 0.0, 0, 0, 0]
          retractTo = pose_sub(contactPose, additionalRetraction)
        end
        movel(retractTo, a=0.02, v=0.1)
        $ 1840 "Until (tool_contact_detection)"
        break
      end
      sync()
    end
    $ 1841 "Direction: Base Z+"
    global move_thread_flag_1841=0
    thread move_thread_1841():
      enter_critical
      move_thread_flag_1841 = 1
      local towardsPos=calculate_point_to_move_towards(p[0.0,0.0,0.0,0.0,0.0,0.0], [0.0,0.0,1.0], 0.08)
      movel(towardsPos, a=0.15, v=0.1)
      move_thread_flag_1841 = 2
      exit_critical
    end
    move_thread_flag_1841 = 0
    move_thread_han_1841 = run move_thread_1841()
    while (True):
      sleep(1.0E-10)
      if (move_thread_flag_1841 > 1):
        join move_thread_han_1841
        $ 1842 "Until (distance)"
        break
      end
      sync()
    end
    $ 1843 "Linea17_B" "breakAfter"
    movel(Linea17_B_p, a=0.5, v=0.1)
    $ 1844 "bajada_comprobacion"
    $ 1845 "Direction: Base Z-"
    global move_thread_flag_1845=0
    thread move_thread_1845():
      enter_critical
      move_thread_flag_1845 = 1
      local towardsPos=calculate_point_to_move_towards(p[0.0,0.0,0.0,0.0,0.0,0.0], [0.0,0.0,-1.0], 0.071)
      movel(towardsPos, a=0.15, v=0.1)
      move_thread_flag_1845 = 2
      exit_critical
    end
    move_thread_flag_1845 = 0
    move_thread_han_1845 = run move_thread_1845()
    while (True):
      sleep(1.0E-10)
      if (move_thread_flag_1845 > 1):
        join move_thread_han_1845
        $ 1846 "Until (distance)"
        break
      end
      sync()
    end
    $ 1847 "Direction: Base Z-"
    global move_thread_flag_1847=0
    thread move_thread_1847():
      enter_critical
      move_thread_flag_1847 = 1
      local towardsPos=calculate_point_to_move_towards(p[0.0,0.0,0.0,0.0,0.0,0.0], [0.0,0.0,-1.0], 1000.0)
      movel(towardsPos, a=0.007, v=0.007)
      move_thread_flag_1847 = 2
      exit_critical
    end
    move_thread_flag_1847 = 0
    move_thread_han_1847 = run move_thread_1847()
    while (True):
      local targetTcpDirection=get_target_tcp_speed()
      local stepsToRetract=tool_contact(direction=targetTcpDirection)
      if (stepsToRetract > 0):
        kill move_thread_han_1847
        stopl(0.02)
        local backTrackMovement=get_actual_joint_positions_history(stepsToRetract)
        local contactPose=get_forward_kin(backTrackMovement)
        local posDir=[targetTcpDirection[0],targetTcpDirection[1],targetTcpDirection[2]]
        local retractTo=contactPose
        if (norm(posDir) > 1e-6):
          local normalizedPosDir=normalize(posDir)
          local additionalRetraction=p[normalizedPosDir[0] * 0.0, normalizedPosDir[1] * 0.0, normalizedPosDir[2] * 0.0, 0, 0, 0]
          retractTo = pose_sub(contactPose, additionalRetraction)
        end
        movel(retractTo, a=0.02, v=0.1)
        $ 1848 "Until (tool_contact_detection)"
        break
      end
      sync()
    end
    $ 1849 "Direction: Base Z+"
    global move_thread_flag_1849=0
    thread move_thread_1849():
      enter_critical
      move_thread_flag_1849 = 1
      local towardsPos=calculate_point_to_move_towards(p[0.0,0.0,0.0,0.0,0.0,0.0], [0.0,0.0,1.0], 0.08)
      movel(towardsPos, a=0.15, v=0.1)
      move_thread_flag_1849 = 2
      exit_critical
    end
    move_thread_flag_1849 = 0
    move_thread_han_1849 = run move_thread_1849()
    while (True):
      sleep(1.0E-10)
      if (move_thread_flag_1849 > 1):
        join move_thread_han_1849
        $ 1850 "Until (distance)"
        break
      end
      sync()
    end
    $ 1851 "AB"
    $ 1852 "'desbaste_inicial'"
    # 'desbaste_inicial'
    $ 1853 "bajada_broca≔p[0,0,-0.008,0,0,0]"
    global bajada_broca=p[0,0,-0.008,0,0,0]
    $ 1854 "barrenos_menos1≔2"
    global barrenos_menos1=2
    $ 1855 "barreno_actual≔0"
    global barreno_actual=0
    $ 1856 "Loop barreno_actual≤barrenos_menos1"
    while (barreno_actual <= barrenos_menos1):
      $ 1857 "Perforacion"
      $ 1858 "MoveL"
      $ 1861 "internos≔interpolate_pose(Linea17_A, Linea17_B, barreno_actual/barrenos_menos1)"
      global internos= interpolate_pose (Linea17_A_p, Linea17_B_p, barreno_actual/barrenos_menos1)
      $ 1862 "internos" "breakAfter"
      movel(internos, a=0.5, v=0.1)
      $ 1863 "'desbaste_inicial'"
      # 'desbaste_inicial'
      $ 1864 "bajada_broca≔p[0,0,-0.024,0,0,0]"
      global bajada_broca=p[0,0,-0.024,0,0,0]
      $ 1865 "bajada≔p[0,0,0.024,0,0,0]"
      global bajada=p[0,0,0.024,0,0,0]
      $ 1866 "Direction: Base Z-"
      global move_thread_flag_1866=0
      thread move_thread_1866():
        enter_critical
        move_thread_flag_1866 = 1
        local towardsPos=calculate_point_to_move_towards(p[0.0,0.0,0.0,0.0,0.0,0.0], [0.0,0.0,-1.0], 0.071)
        movel(towardsPos, a=0.15, v=0.1)
        move_thread_flag_1866 = 2
        exit_critical
      end
      move_thread_flag_1866 = 0
      move_thread_han_1866 = run move_thread_1866()
      while (True):
        sleep(1.0E-10)
        if (move_thread_flag_1866 > 1):
          join move_thread_han_1866
          $ 1867 "Until (distance)"
          break
        end
        sync()
      end
      $ 1868 "Direction: Base Z-"
      global move_thread_flag_1868=0
      thread move_thread_1868():
        enter_critical
        move_thread_flag_1868 = 1
        local towardsPos=calculate_point_to_move_towards(p[0.0,0.0,0.0,0.0,0.0,0.0], [0.0,0.0,-1.0], 1000.0)
        movel(towardsPos, a=0.007, v=0.007)
        move_thread_flag_1868 = 2
        exit_critical
      end
      move_thread_flag_1868 = 0
      move_thread_han_1868 = run move_thread_1868()
      while (True):
        local targetTcpDirection=get_target_tcp_speed()
        local stepsToRetract=tool_contact(direction=targetTcpDirection)
        if (stepsToRetract > 0):
          kill move_thread_han_1868
          stopl(0.02)
          local backTrackMovement=get_actual_joint_positions_history(stepsToRetract)
          local contactPose=get_forward_kin(backTrackMovement)
          local posDir=[targetTcpDirection[0],targetTcpDirection[1],targetTcpDirection[2]]
          local retractTo=contactPose
          if (norm(posDir) > 1e-6):
            local normalizedPosDir=normalize(posDir)
            local additionalRetraction=p[normalizedPosDir[0] * 0.0, normalizedPosDir[1] * 0.0, normalizedPosDir[2] * 0.0, 0, 0, 0]
            retractTo = pose_sub(contactPose, additionalRetraction)
          end
          movel(retractTo, a=0.02, v=0.1)
          $ 1869 "Until (tool_contact_detection)"
          break
        end
        sync()
      end
      $ 1870 "Popup: punto contacto alanzdo"
      popup("punto contacto alanzdo", "Mensaje", False, False, blocking=True)
      $ 1871 "Direction: Base Z+"
      global move_thread_flag_1871=0
      thread move_thread_1871():
        enter_critical
        move_thread_flag_1871 = 1
        local towardsPos=calculate_point_to_move_towards(p[0.0,0.0,0.0,0.0,0.0,0.0], [0.0,0.0,1.0], 0.002)
        movel(towardsPos, a=0.15, v=0.1)
        move_thread_flag_1871 = 2
        exit_critical
      end
      move_thread_flag_1871 = 0
      move_thread_han_1871 = run move_thread_1871()
      while (True):
        sleep(1.0E-10)
        if (move_thread_flag_1871 > 1):
          join move_thread_han_1871
          $ 1872 "Until (distance)"
          break
        end
        sync()
      end
      $ 1873 "Wait: 0.3"
      sleep(0.3)
      $ 1874 "Set CO[1]=Encender"
      set_configurable_digital_out(1, True)
      $ 1875 "Wait: 0.3"
      sleep(0.3)
      $ 1876 "Loop 1 times"
      Loop_137 = 0
      while (Loop_137 < 1):
        $ 1877 "bajar≔pose_add(get_actual_tcp_pose(), bajada_broca)"
        global bajar= pose_add ( get_actual_tcp_pose (), bajada_broca)
        $ 1878 "bajar" "breakAfter"
        movel(bajar, a=0.004, v=0.004)
        $ 1879 "subir≔pose_sub(get_actual_tcp_pose(), bajada_broca)"
        global subir= pose_sub ( get_actual_tcp_pose (), bajada_broca)
        $ 1880 "Direction: Base Z+"
        global move_thread_flag_1880=0
        thread move_thread_1880():
          enter_critical
          move_thread_flag_1880 = 1
          local towardsPos=calculate_point_to_move_towards(p[0.0,0.0,0.0,0.0,0.0,0.0], [0.0,0.0,1.0], 0.002)
          movel(towardsPos, a=0.015, v=0.015)
          move_thread_flag_1880 = 2
          exit_critical
        end
        move_thread_flag_1880 = 0
        move_thread_han_1880 = run move_thread_1880()
        while (True):
          sleep(1.0E-10)
          if (move_thread_flag_1880 > 1):
            join move_thread_han_1880
            $ 1881 "Until (distance)"
            break
          end
          sync()
        end
        $ 1882 "Set CO[1]=Apagar"
        set_configurable_digital_out(1, False)
        $ 1883 "subir" "breakAfter"
        movel(subir, a=0.015, v=0.015)
        $ 1884 "bajada_broca≔pose_sub(bajada_broca, bajada)"
        global bajada_broca= pose_sub (bajada_broca, bajada)
        Loop_137 = Loop_137 + 1
      end
      $ 1885 "Direction: Base Z+"
      global move_thread_flag_1885=0
      thread move_thread_1885():
        enter_critical
        move_thread_flag_1885 = 1
        local towardsPos=calculate_point_to_move_towards(p[0.0,0.0,0.0,0.0,0.0,0.0], [0.0,0.0,1.0], 0.08)
        movel(towardsPos, a=0.035, v=0.03)
        move_thread_flag_1885 = 2
        exit_critical
      end
      move_thread_flag_1885 = 0
      move_thread_han_1885 = run move_thread_1885()
      while (True):
        sleep(1.0E-10)
        if (move_thread_flag_1885 > 1):
          join move_thread_han_1885
          $ 1886 "Until (distance)"
          break
        end
        sync()
      end
      $ 1887 "Set CO[1]=Apagar"
      set_configurable_digital_out(1, False)
      $ 1888 "barreno_actual≔barreno_actual+1"
      global barreno_actual=barreno_actual+1
    end
    $ 1891 "Popup: Linea17 con chica Terminada!"
    popup("Linea17 con chica Terminada!", "Mensaje", False, False, blocking=True)
    $ 1892 "Linea18"
    $ 1893 "Marcar_puntos"
    $ 1894 "MoveL"
    $ 1895 "Linea18_A" "breakAfter"
    movel(Linea18_A_p, a=0.5, v=0.1)
    $ 1896 "bajada_comprobacion"
    $ 1897 "Direction: Base Z-"
    global move_thread_flag_1897=0
    thread move_thread_1897():
      enter_critical
      move_thread_flag_1897 = 1
      local towardsPos=calculate_point_to_move_towards(p[0.0,0.0,0.0,0.0,0.0,0.0], [0.0,0.0,-1.0], 0.071)
      movel(towardsPos, a=0.15, v=0.1)
      move_thread_flag_1897 = 2
      exit_critical
    end
    move_thread_flag_1897 = 0
    move_thread_han_1897 = run move_thread_1897()
    while (True):
      sleep(1.0E-10)
      if (move_thread_flag_1897 > 1):
        join move_thread_han_1897
        $ 1898 "Until (distance)"
        break
      end
      sync()
    end
    $ 1899 "Direction: Base Z-"
    global move_thread_flag_1899=0
    thread move_thread_1899():
      enter_critical
      move_thread_flag_1899 = 1
      local towardsPos=calculate_point_to_move_towards(p[0.0,0.0,0.0,0.0,0.0,0.0], [0.0,0.0,-1.0], 1000.0)
      movel(towardsPos, a=0.007, v=0.007)
      move_thread_flag_1899 = 2
      exit_critical
    end
    move_thread_flag_1899 = 0
    move_thread_han_1899 = run move_thread_1899()
    while (True):
      local targetTcpDirection=get_target_tcp_speed()
      local stepsToRetract=tool_contact(direction=targetTcpDirection)
      if (stepsToRetract > 0):
        kill move_thread_han_1899
        stopl(0.02)
        local backTrackMovement=get_actual_joint_positions_history(stepsToRetract)
        local contactPose=get_forward_kin(backTrackMovement)
        local posDir=[targetTcpDirection[0],targetTcpDirection[1],targetTcpDirection[2]]
        local retractTo=contactPose
        if (norm(posDir) > 1e-6):
          local normalizedPosDir=normalize(posDir)
          local additionalRetraction=p[normalizedPosDir[0] * 0.0, normalizedPosDir[1] * 0.0, normalizedPosDir[2] * 0.0, 0, 0, 0]
          retractTo = pose_sub(contactPose, additionalRetraction)
        end
        movel(retractTo, a=0.02, v=0.1)
        $ 1900 "Until (tool_contact_detection)"
        break
      end
      sync()
    end
    $ 1901 "Direction: Base Z+"
    global move_thread_flag_1901=0
    thread move_thread_1901():
      enter_critical
      move_thread_flag_1901 = 1
      local towardsPos=calculate_point_to_move_towards(p[0.0,0.0,0.0,0.0,0.0,0.0], [0.0,0.0,1.0], 0.08)
      movel(towardsPos, a=0.15, v=0.1)
      move_thread_flag_1901 = 2
      exit_critical
    end
    move_thread_flag_1901 = 0
    move_thread_han_1901 = run move_thread_1901()
    while (True):
      sleep(1.0E-10)
      if (move_thread_flag_1901 > 1):
        join move_thread_han_1901
        $ 1902 "Until (distance)"
        break
      end
      sync()
    end
    $ 1903 "Linea18_AB" "breakAfter"
    movel(Linea18_AB_p, a=0.5, v=0.1)
    $ 1905 "bajada_comprobacion"
    $ 1906 "Direction: Base Z-"
    global move_thread_flag_1906=0
    thread move_thread_1906():
      enter_critical
      move_thread_flag_1906 = 1
      local towardsPos=calculate_point_to_move_towards(p[0.0,0.0,0.0,0.0,0.0,0.0], [0.0,0.0,-1.0], 0.071)
      movel(towardsPos, a=0.15, v=0.1)
      move_thread_flag_1906 = 2
      exit_critical
    end
    move_thread_flag_1906 = 0
    move_thread_han_1906 = run move_thread_1906()
    while (True):
      sleep(1.0E-10)
      if (move_thread_flag_1906 > 1):
        join move_thread_han_1906
        $ 1907 "Until (distance)"
        break
      end
      sync()
    end
    $ 1908 "Direction: Base Z-"
    global move_thread_flag_1908=0
    thread move_thread_1908():
      enter_critical
      move_thread_flag_1908 = 1
      local towardsPos=calculate_point_to_move_towards(p[0.0,0.0,0.0,0.0,0.0,0.0], [0.0,0.0,-1.0], 1000.0)
      movel(towardsPos, a=0.007, v=0.007)
      move_thread_flag_1908 = 2
      exit_critical
    end
    move_thread_flag_1908 = 0
    move_thread_han_1908 = run move_thread_1908()
    while (True):
      local targetTcpDirection=get_target_tcp_speed()
      local stepsToRetract=tool_contact(direction=targetTcpDirection)
      if (stepsToRetract > 0):
        kill move_thread_han_1908
        stopl(0.02)
        local backTrackMovement=get_actual_joint_positions_history(stepsToRetract)
        local contactPose=get_forward_kin(backTrackMovement)
        local posDir=[targetTcpDirection[0],targetTcpDirection[1],targetTcpDirection[2]]
        local retractTo=contactPose
        if (norm(posDir) > 1e-6):
          local normalizedPosDir=normalize(posDir)
          local additionalRetraction=p[normalizedPosDir[0] * 0.0, normalizedPosDir[1] * 0.0, normalizedPosDir[2] * 0.0, 0, 0, 0]
          retractTo = pose_sub(contactPose, additionalRetraction)
        end
        movel(retractTo, a=0.02, v=0.1)
        $ 1909 "Until (tool_contact_detection)"
        break
      end
      sync()
    end
    $ 1910 "Direction: Base Z+"
    global move_thread_flag_1910=0
    thread move_thread_1910():
      enter_critical
      move_thread_flag_1910 = 1
      local towardsPos=calculate_point_to_move_towards(p[0.0,0.0,0.0,0.0,0.0,0.0], [0.0,0.0,1.0], 0.08)
      movel(towardsPos, a=0.15, v=0.1)
      move_thread_flag_1910 = 2
      exit_critical
    end
    move_thread_flag_1910 = 0
    move_thread_han_1910 = run move_thread_1910()
    while (True):
      sleep(1.0E-10)
      if (move_thread_flag_1910 > 1):
        join move_thread_han_1910
        $ 1911 "Until (distance)"
        break
      end
      sync()
    end
    $ 1912 "AB"
    $ 1913 "'desbaste_inicial'"
    # 'desbaste_inicial'
    $ 1914 "bajada_broca≔p[0,0,-0.008,0,0,0]"
    global bajada_broca=p[0,0,-0.008,0,0,0]
    $ 1915 "barrenos_menos1≔9"
    global barrenos_menos1=9
    $ 1916 "barreno_actual≔0"
    global barreno_actual=0
    $ 1917 "Loop barreno_actual≤barrenos_menos1"
    while (barreno_actual <= barrenos_menos1):
      $ 1918 "Perforacion"
      $ 1919 "MoveL"
      $ 1920 "If barreno_actual≟6 "
      if (barreno_actual == 6 ):
        $ 1921 "barreno_actual≔barreno_actual+1"
        global barreno_actual=barreno_actual+1
      end
      $ 1922 "internos≔interpolate_pose(Linea18_A, Linea18_AB, barreno_actual/barrenos_menos1)"
      global internos= interpolate_pose (Linea18_A_p, Linea18_AB_p, barreno_actual/barrenos_menos1)
      $ 1923 "internos" "breakAfter"
      movel(internos, a=0.5, v=0.1)
      $ 1924 "'desbaste_inicial'"
      # 'desbaste_inicial'
      $ 1925 "bajada_broca≔p[0,0,-0.024,0,0,0]"
      global bajada_broca=p[0,0,-0.024,0,0,0]
      $ 1926 "bajada≔p[0,0,0.024,0,0,0]"
      global bajada=p[0,0,0.024,0,0,0]
      $ 1927 "Direction: Base Z-"
      global move_thread_flag_1927=0
      thread move_thread_1927():
        enter_critical
        move_thread_flag_1927 = 1
        local towardsPos=calculate_point_to_move_towards(p[0.0,0.0,0.0,0.0,0.0,0.0], [0.0,0.0,-1.0], 0.071)
        movel(towardsPos, a=0.15, v=0.1)
        move_thread_flag_1927 = 2
        exit_critical
      end
      move_thread_flag_1927 = 0
      move_thread_han_1927 = run move_thread_1927()
      while (True):
        sleep(1.0E-10)
        if (move_thread_flag_1927 > 1):
          join move_thread_han_1927
          $ 1928 "Until (distance)"
          break
        end
        sync()
      end
      $ 1929 "Direction: Base Z-"
      global move_thread_flag_1929=0
      thread move_thread_1929():
        enter_critical
        move_thread_flag_1929 = 1
        local towardsPos=calculate_point_to_move_towards(p[0.0,0.0,0.0,0.0,0.0,0.0], [0.0,0.0,-1.0], 1000.0)
        movel(towardsPos, a=0.007, v=0.007)
        move_thread_flag_1929 = 2
        exit_critical
      end
      move_thread_flag_1929 = 0
      move_thread_han_1929 = run move_thread_1929()
      while (True):
        local targetTcpDirection=get_target_tcp_speed()
        local stepsToRetract=tool_contact(direction=targetTcpDirection)
        if (stepsToRetract > 0):
          kill move_thread_han_1929
          stopl(0.02)
          local backTrackMovement=get_actual_joint_positions_history(stepsToRetract)
          local contactPose=get_forward_kin(backTrackMovement)
          local posDir=[targetTcpDirection[0],targetTcpDirection[1],targetTcpDirection[2]]
          local retractTo=contactPose
          if (norm(posDir) > 1e-6):
            local normalizedPosDir=normalize(posDir)
            local additionalRetraction=p[normalizedPosDir[0] * 0.0, normalizedPosDir[1] * 0.0, normalizedPosDir[2] * 0.0, 0, 0, 0]
            retractTo = pose_sub(contactPose, additionalRetraction)
          end
          movel(retractTo, a=0.02, v=0.1)
          $ 1930 "Until (tool_contact_detection)"
          break
        end
        sync()
      end
      $ 1931 "Popup: punto contacto alanzdo"
      popup("punto contacto alanzdo", "Mensaje", False, False, blocking=True)
      $ 1932 "Direction: Base Z+"
      global move_thread_flag_1932=0
      thread move_thread_1932():
        enter_critical
        move_thread_flag_1932 = 1
        local towardsPos=calculate_point_to_move_towards(p[0.0,0.0,0.0,0.0,0.0,0.0], [0.0,0.0,1.0], 0.007)
        movel(towardsPos, a=0.015, v=0.015)
        move_thread_flag_1932 = 2
        exit_critical
      end
      move_thread_flag_1932 = 0
      move_thread_han_1932 = run move_thread_1932()
      while (True):
        sleep(1.0E-10)
        if (move_thread_flag_1932 > 1):
          join move_thread_han_1932
          $ 1933 "Until (distance)"
          break
        end
        sync()
      end
      $ 1934 "Wait: 0.3"
      sleep(0.3)
      $ 1935 "Set CO[1]=Encender"
      set_configurable_digital_out(1, True)
      $ 1936 "Wait: 0.3"
      sleep(0.3)
      $ 1937 "Loop 1 times"
      Loop_139 = 0
      while (Loop_139 < 1):
        $ 1938 "bajar≔pose_add(get_actual_tcp_pose(), bajada_broca)"
        global bajar= pose_add ( get_actual_tcp_pose (), bajada_broca)
        $ 1939 "bajar" "breakAfter"
        movel(bajar, a=0.004, v=0.004)
        $ 1940 "subir≔pose_sub(get_actual_tcp_pose(), bajada_broca)"
        global subir= pose_sub ( get_actual_tcp_pose (), bajada_broca)
        $ 1941 "Direction: Base Z+"
        global move_thread_flag_1941=0
        thread move_thread_1941():
          enter_critical
          move_thread_flag_1941 = 1
          local towardsPos=calculate_point_to_move_towards(p[0.0,0.0,0.0,0.0,0.0,0.0], [0.0,0.0,1.0], 0.002)
          movel(towardsPos, a=0.015, v=0.015)
          move_thread_flag_1941 = 2
          exit_critical
        end
        move_thread_flag_1941 = 0
        move_thread_han_1941 = run move_thread_1941()
        while (True):
          sleep(1.0E-10)
          if (move_thread_flag_1941 > 1):
            join move_thread_han_1941
            $ 1942 "Until (distance)"
            break
          end
          sync()
        end
        $ 1943 "Set CO[1]=Apagar"
        set_configurable_digital_out(1, False)
        $ 1944 "subir" "breakAfter"
        movel(subir, a=0.015, v=0.015)
        $ 1945 "bajada_broca≔pose_sub(bajada_broca, bajada)"
        global bajada_broca= pose_sub (bajada_broca, bajada)
        Loop_139 = Loop_139 + 1
      end
      $ 1946 "Direction: Base Z+"
      global move_thread_flag_1946=0
      thread move_thread_1946():
        enter_critical
        move_thread_flag_1946 = 1
        local towardsPos=calculate_point_to_move_towards(p[0.0,0.0,0.0,0.0,0.0,0.0], [0.0,0.0,1.0], 0.08)
        movel(towardsPos, a=0.15, v=0.1)
        move_thread_flag_1946 = 2
        exit_critical
      end
      move_thread_flag_1946 = 0
      move_thread_han_1946 = run move_thread_1946()
      while (True):
        sleep(1.0E-10)
        if (move_thread_flag_1946 > 1):
          join move_thread_han_1946
          $ 1947 "Until (distance)"
          break
        end
        sync()
      end
      $ 1948 "Set CO[1]=Apagar"
      set_configurable_digital_out(1, False)
      $ 1949 "barreno_actual≔barreno_actual+1"
      global barreno_actual=barreno_actual+1
    end
    $ 1952 "Popup: Linea18 con chica Terminada!"
    popup("Linea18 con chica Terminada!", "Mensaje", False, False, blocking=True)
    $ 1953 "Linea18B"
    $ 1954 "Marcar_puntos"
    $ 1955 "MoveL"
    $ 1956 "Linea18_BA" "breakAfter"
    movel(Linea18_BA_p, a=0.5, v=0.1)
    $ 1957 "bajada_comprobacion"
    $ 1958 "Direction: Base Z-"
    global move_thread_flag_1958=0
    thread move_thread_1958():
      enter_critical
      move_thread_flag_1958 = 1
      local towardsPos=calculate_point_to_move_towards(p[0.0,0.0,0.0,0.0,0.0,0.0], [0.0,0.0,-1.0], 0.071)
      movel(towardsPos, a=0.15, v=0.1)
      move_thread_flag_1958 = 2
      exit_critical
    end
    move_thread_flag_1958 = 0
    move_thread_han_1958 = run move_thread_1958()
    while (True):
      sleep(1.0E-10)
      if (move_thread_flag_1958 > 1):
        join move_thread_han_1958
        $ 1959 "Until (distance)"
        break
      end
      sync()
    end
    $ 1960 "Direction: Base Z-"
    global move_thread_flag_1960=0
    thread move_thread_1960():
      enter_critical
      move_thread_flag_1960 = 1
      local towardsPos=calculate_point_to_move_towards(p[0.0,0.0,0.0,0.0,0.0,0.0], [0.0,0.0,-1.0], 1000.0)
      movel(towardsPos, a=0.007, v=0.007)
      move_thread_flag_1960 = 2
      exit_critical
    end
    move_thread_flag_1960 = 0
    move_thread_han_1960 = run move_thread_1960()
    while (True):
      local targetTcpDirection=get_target_tcp_speed()
      local stepsToRetract=tool_contact(direction=targetTcpDirection)
      if (stepsToRetract > 0):
        kill move_thread_han_1960
        stopl(0.02)
        local backTrackMovement=get_actual_joint_positions_history(stepsToRetract)
        local contactPose=get_forward_kin(backTrackMovement)
        local posDir=[targetTcpDirection[0],targetTcpDirection[1],targetTcpDirection[2]]
        local retractTo=contactPose
        if (norm(posDir) > 1e-6):
          local normalizedPosDir=normalize(posDir)
          local additionalRetraction=p[normalizedPosDir[0] * 0.0, normalizedPosDir[1] * 0.0, normalizedPosDir[2] * 0.0, 0, 0, 0]
          retractTo = pose_sub(contactPose, additionalRetraction)
        end
        movel(retractTo, a=0.02, v=0.1)
        $ 1961 "Until (tool_contact_detection)"
        break
      end
      sync()
    end
    $ 1962 "Direction: Base Z+"
    global move_thread_flag_1962=0
    thread move_thread_1962():
      enter_critical
      move_thread_flag_1962 = 1
      local towardsPos=calculate_point_to_move_towards(p[0.0,0.0,0.0,0.0,0.0,0.0], [0.0,0.0,1.0], 0.08)
      movel(towardsPos, a=0.15, v=0.1)
      move_thread_flag_1962 = 2
      exit_critical
    end
    move_thread_flag_1962 = 0
    move_thread_han_1962 = run move_thread_1962()
    while (True):
      sleep(1.0E-10)
      if (move_thread_flag_1962 > 1):
        join move_thread_han_1962
        $ 1963 "Until (distance)"
        break
      end
      sync()
    end
    $ 1965 "Linea18_B" "breakAfter"
    movel(Linea18_B_p, a=0.5, v=0.1)
    $ 1966 "bajada_comprobacion"
    $ 1967 "Direction: Base Z-"
    global move_thread_flag_1967=0
    thread move_thread_1967():
      enter_critical
      move_thread_flag_1967 = 1
      local towardsPos=calculate_point_to_move_towards(p[0.0,0.0,0.0,0.0,0.0,0.0], [0.0,0.0,-1.0], 0.071)
      movel(towardsPos, a=0.15, v=0.1)
      move_thread_flag_1967 = 2
      exit_critical
    end
    move_thread_flag_1967 = 0
    move_thread_han_1967 = run move_thread_1967()
    while (True):
      sleep(1.0E-10)
      if (move_thread_flag_1967 > 1):
        join move_thread_han_1967
        $ 1968 "Until (distance)"
        break
      end
      sync()
    end
    $ 1969 "Direction: Base Z-"
    global move_thread_flag_1969=0
    thread move_thread_1969():
      enter_critical
      move_thread_flag_1969 = 1
      local towardsPos=calculate_point_to_move_towards(p[0.0,0.0,0.0,0.0,0.0,0.0], [0.0,0.0,-1.0], 1000.0)
      movel(towardsPos, a=0.007, v=0.007)
      move_thread_flag_1969 = 2
      exit_critical
    end
    move_thread_flag_1969 = 0
    move_thread_han_1969 = run move_thread_1969()
    while (True):
      local targetTcpDirection=get_target_tcp_speed()
      local stepsToRetract=tool_contact(direction=targetTcpDirection)
      if (stepsToRetract > 0):
        kill move_thread_han_1969
        stopl(0.02)
        local backTrackMovement=get_actual_joint_positions_history(stepsToRetract)
        local contactPose=get_forward_kin(backTrackMovement)
        local posDir=[targetTcpDirection[0],targetTcpDirection[1],targetTcpDirection[2]]
        local retractTo=contactPose
        if (norm(posDir) > 1e-6):
          local normalizedPosDir=normalize(posDir)
          local additionalRetraction=p[normalizedPosDir[0] * 0.0, normalizedPosDir[1] * 0.0, normalizedPosDir[2] * 0.0, 0, 0, 0]
          retractTo = pose_sub(contactPose, additionalRetraction)
        end
        movel(retractTo, a=0.02, v=0.1)
        $ 1970 "Until (tool_contact_detection)"
        break
      end
      sync()
    end
    $ 1971 "Direction: Base Z+"
    global move_thread_flag_1971=0
    thread move_thread_1971():
      enter_critical
      move_thread_flag_1971 = 1
      local towardsPos=calculate_point_to_move_towards(p[0.0,0.0,0.0,0.0,0.0,0.0], [0.0,0.0,1.0], 0.08)
      movel(towardsPos, a=0.15, v=0.1)
      move_thread_flag_1971 = 2
      exit_critical
    end
    move_thread_flag_1971 = 0
    move_thread_han_1971 = run move_thread_1971()
    while (True):
      sleep(1.0E-10)
      if (move_thread_flag_1971 > 1):
        join move_thread_han_1971
        $ 1972 "Until (distance)"
        break
      end
      sync()
    end
    $ 1973 "AB"
    $ 1974 "'desbaste_inicial'"
    # 'desbaste_inicial'
    $ 1975 "bajada_broca≔p[0,0,-0.008,0,0,0]"
    global bajada_broca=p[0,0,-0.008,0,0,0]
    $ 1976 "barrenos_menos1≔9"
    global barrenos_menos1=9
    $ 1977 "barreno_actual≔0"
    global barreno_actual=0
    $ 1978 "Loop barreno_actual≤barrenos_menos1"
    while (barreno_actual <= barrenos_menos1):
      $ 1979 "Perforacion"
      $ 1980 "MoveL"
      $ 1981 "If barreno_actual≟3"
      if (barreno_actual == 3):
        $ 1982 "barreno_actual≔barreno_actual+1"
        global barreno_actual=barreno_actual+1
      end
      $ 1983 "internos≔interpolate_pose(Linea18_BA, Linea18_B, barreno_actual/barrenos_menos1)"
      global internos= interpolate_pose (Linea18_BA_p, Linea18_B_p, barreno_actual/barrenos_menos1)
      $ 1984 "internos" "breakAfter"
      movel(internos, a=0.5, v=0.1)
      $ 1985 "'desbaste_inicial'"
      # 'desbaste_inicial'
      $ 1986 "bajada_broca≔p[0,0,-0.024,0,0,0]"
      global bajada_broca=p[0,0,-0.024,0,0,0]
      $ 1987 "bajada≔p[0,0,0.024,0,0,0]"
      global bajada=p[0,0,0.024,0,0,0]
      $ 1988 "Direction: Base Z-"
      global move_thread_flag_1988=0
      thread move_thread_1988():
        enter_critical
        move_thread_flag_1988 = 1
        local towardsPos=calculate_point_to_move_towards(p[0.0,0.0,0.0,0.0,0.0,0.0], [0.0,0.0,-1.0], 0.071)
        movel(towardsPos, a=0.15, v=0.1)
        move_thread_flag_1988 = 2
        exit_critical
      end
      move_thread_flag_1988 = 0
      move_thread_han_1988 = run move_thread_1988()
      while (True):
        sleep(1.0E-10)
        if (move_thread_flag_1988 > 1):
          join move_thread_han_1988
          $ 1989 "Until (distance)"
          break
        end
        sync()
      end
      $ 1990 "Direction: Base Z-"
      global move_thread_flag_1990=0
      thread move_thread_1990():
        enter_critical
        move_thread_flag_1990 = 1
        local towardsPos=calculate_point_to_move_towards(p[0.0,0.0,0.0,0.0,0.0,0.0], [0.0,0.0,-1.0], 1000.0)
        movel(towardsPos, a=0.007, v=0.007)
        move_thread_flag_1990 = 2
        exit_critical
      end
      move_thread_flag_1990 = 0
      move_thread_han_1990 = run move_thread_1990()
      while (True):
        local targetTcpDirection=get_target_tcp_speed()
        local stepsToRetract=tool_contact(direction=targetTcpDirection)
        if (stepsToRetract > 0):
          kill move_thread_han_1990
          stopl(0.02)
          local backTrackMovement=get_actual_joint_positions_history(stepsToRetract)
          local contactPose=get_forward_kin(backTrackMovement)
          local posDir=[targetTcpDirection[0],targetTcpDirection[1],targetTcpDirection[2]]
          local retractTo=contactPose
          if (norm(posDir) > 1e-6):
            local normalizedPosDir=normalize(posDir)
            local additionalRetraction=p[normalizedPosDir[0] * 0.0, normalizedPosDir[1] * 0.0, normalizedPosDir[2] * 0.0, 0, 0, 0]
            retractTo = pose_sub(contactPose, additionalRetraction)
          end
          movel(retractTo, a=0.02, v=0.1)
          $ 1991 "Until (tool_contact_detection)"
          break
        end
        sync()
      end
      $ 1992 "Popup: punto contacto alanzdo"
      popup("punto contacto alanzdo", "Mensaje", False, False, blocking=True)
      $ 1993 "Direction: Base Z+"
      global move_thread_flag_1993=0
      thread move_thread_1993():
        enter_critical
        move_thread_flag_1993 = 1
        local towardsPos=calculate_point_to_move_towards(p[0.0,0.0,0.0,0.0,0.0,0.0], [0.0,0.0,1.0], 0.007)
        movel(towardsPos, a=0.015, v=0.015)
        move_thread_flag_1993 = 2
        exit_critical
      end
      move_thread_flag_1993 = 0
      move_thread_han_1993 = run move_thread_1993()
      while (True):
        sleep(1.0E-10)
        if (move_thread_flag_1993 > 1):
          join move_thread_han_1993
          $ 1994 "Until (distance)"
          break
        end
        sync()
      end
      $ 1995 "Wait: 0.3"
      sleep(0.3)
      $ 1996 "Set CO[1]=Encender"
      set_configurable_digital_out(1, True)
      $ 1997 "Wait: 0.3"
      sleep(0.3)
      $ 1998 "Loop 1 times"
      Loop_28 = 0
      while (Loop_28 < 1):
        $ 1999 "bajar≔pose_add(get_actual_tcp_pose(), bajada_broca)"
        global bajar= pose_add ( get_actual_tcp_pose (), bajada_broca)
        $ 2000 "bajar" "breakAfter"
        movel(bajar, a=0.004, v=0.004)
        $ 2001 "subir≔pose_sub(get_actual_tcp_pose(), bajada_broca)"
        global subir= pose_sub ( get_actual_tcp_pose (), bajada_broca)
        $ 2002 "Direction: Base Z+"
        global move_thread_flag_2002=0
        thread move_thread_2002():
          enter_critical
          move_thread_flag_2002 = 1
          local towardsPos=calculate_point_to_move_towards(p[0.0,0.0,0.0,0.0,0.0,0.0], [0.0,0.0,1.0], 0.002)
          movel(towardsPos, a=0.015, v=0.015)
          move_thread_flag_2002 = 2
          exit_critical
        end
        move_thread_flag_2002 = 0
        move_thread_han_2002 = run move_thread_2002()
        while (True):
          sleep(1.0E-10)
          if (move_thread_flag_2002 > 1):
            join move_thread_han_2002
            $ 2003 "Until (distance)"
            break
          end
          sync()
        end
        $ 2004 "Set CO[1]=Apagar"
        set_configurable_digital_out(1, False)
        $ 2005 "subir" "breakAfter"
        movel(subir, a=0.015, v=0.015)
        $ 2006 "bajada_broca≔pose_sub(bajada_broca, bajada)"
        global bajada_broca= pose_sub (bajada_broca, bajada)
        Loop_28 = Loop_28 + 1
      end
      $ 2007 "Direction: Base Z+"
      global move_thread_flag_2007=0
      thread move_thread_2007():
        enter_critical
        move_thread_flag_2007 = 1
        local towardsPos=calculate_point_to_move_towards(p[0.0,0.0,0.0,0.0,0.0,0.0], [0.0,0.0,1.0], 0.08)
        movel(towardsPos, a=0.15, v=0.1)
        move_thread_flag_2007 = 2
        exit_critical
      end
      move_thread_flag_2007 = 0
      move_thread_han_2007 = run move_thread_2007()
      while (True):
        sleep(1.0E-10)
        if (move_thread_flag_2007 > 1):
          join move_thread_han_2007
          $ 2008 "Until (distance)"
          break
        end
        sync()
      end
      $ 2009 "Set CO[1]=Apagar"
      set_configurable_digital_out(1, False)
      $ 2010 "barreno_actual≔barreno_actual+1"
      global barreno_actual=barreno_actual+1
    end
    $ 2013 "Popup: Linea18B con chica Terminada!"
    popup("Linea18B con chica Terminada!", "Mensaje", False, False, blocking=True)
    $ 2014 "cambiar_broca≔ True "
    global cambiar_broca=  True
    $ 2015 "Call Quitar_broca"
    Quitar_broca()
    $ 2016 "Call Poner_broca"
    Poner_broca()
    $ 3183 "Posicion3"
    $ 3184 "Inicio"
    $ 3185 "eje7≔3"
    global eje7=3
    $ 3186 "MoveL"
    $ 3187 "Home3" "breakAfter"
    movel(Home3_p, a=1.2, v=0.25)
    $ 3188 "SeatTracks"
    $ 3189 "Broca_1"
    $ 3190 "Linea3"
    $ 3191 "Marcar_puntos"
    $ 3192 "MoveL"
    $ 3193 "Home3" "breakAfter"
    movel(Home3_p, a=0.5, v=0.1)
    $ 3200 "Linea3_A" "breakAfter"
    movel(Linea3_A_p, a=0.5, v=0.1)
    $ 3201 "Linea3_B" "breakAfter"
    movel(Linea3_B_p, a=0.5, v=0.1)
    $ 3202 "Linea3_C" "breakAfter"
    movel(Linea3_C_p, a=0.5, v=0.1)
    $ 3203 "Linea3_D" "breakAfter"
    movel(Linea3_D_p, a=0.5, v=0.1)
    $ 3204 "Linea3_E" "breakAfter"
    movel(Linea3_E_p, a=0.5, v=0.1)
    $ 3205 "Linea3_F" "breakAfter"
    movel(Linea3_F_p, a=0.5, v=0.1)
    $ 3206 "AB"
    $ 3207 "'desbaste_inicial'"
    # 'desbaste_inicial'
    $ 3208 "bajada_broca≔p[0,0,-0.008,0,0,0]"
    global bajada_broca=p[0,0,-0.008,0,0,0]
    $ 3209 "barrenos_menos1≔8"
    global barrenos_menos1=8
    $ 3210 "barreno_actual≔0"
    global barreno_actual=0
    $ 3211 "Loop barreno_actual≤barrenos_menos1"
    while (barreno_actual <= barrenos_menos1):
      $ 3212 "Perforacion"
      $ 3213 "MoveL"
      $ 3214 "internos≔interpolate_pose(Linea3_A, Linea3_B, barreno_actual/barrenos_menos1)"
      global internos= interpolate_pose (Linea3_A_p, Linea3_B_p, barreno_actual/barrenos_menos1)
      $ 3215 "internos" "breakAfter"
      movel(internos, a=0.5, v=0.1)
      $ 3216 "'desbaste_inicial'"
      # 'desbaste_inicial'
      $ 3217 "bajada_broca≔p[0,0,-0.008,0,0,0]"
      global bajada_broca=p[0,0,-0.008,0,0,0]
      $ 3218 "bajada≔p[0,0,0.008,0,0,0]"
      global bajada=p[0,0,0.008,0,0,0]
      $ 3219 "Direction: Base Z-"
      global move_thread_flag_3219=0
      thread move_thread_3219():
        enter_critical
        move_thread_flag_3219 = 1
        local towardsPos=calculate_point_to_move_towards(p[0.0,0.0,0.0,0.0,0.0,0.0], [0.0,0.0,-1.0], 0.08)
        movel(towardsPos, a=0.035, v=0.03)
        move_thread_flag_3219 = 2
        exit_critical
      end
      move_thread_flag_3219 = 0
      move_thread_han_3219 = run move_thread_3219()
      while (True):
        sleep(1.0E-10)
        if (move_thread_flag_3219 > 1):
          join move_thread_han_3219
          $ 3220 "Until (distance)"
          break
        end
        sync()
      end
      $ 3221 "Popup: punto contacto alanzdo"
      popup("punto contacto alanzdo", "Mensaje", False, False, blocking=True)
      $ 3222 "Direction: Base Z+"
      global move_thread_flag_3222=0
      thread move_thread_3222():
        enter_critical
        move_thread_flag_3222 = 1
        local towardsPos=calculate_point_to_move_towards(p[0.0,0.0,0.0,0.0,0.0,0.0], [0.0,0.0,1.0], 0.002)
        movel(towardsPos, a=0.005, v=0.003)
        move_thread_flag_3222 = 2
        exit_critical
      end
      move_thread_flag_3222 = 0
      move_thread_han_3222 = run move_thread_3222()
      while (True):
        sleep(1.0E-10)
        if (move_thread_flag_3222 > 1):
          join move_thread_han_3222
          $ 3223 "Until (distance)"
          break
        end
        sync()
      end
      $ 3224 "Wait: 0.3"
      sleep(0.3)
      $ 3225 "Set CO[1]=Encender"
      set_configurable_digital_out(1, True)
      $ 3226 "Wait: 0.3"
      sleep(0.3)
      $ 3227 "Loop 3 times"
      Loop_21 = 0
      while (Loop_21 < 3):
        $ 3228 "bajar≔pose_add(get_actual_tcp_pose(), bajada_broca)"
        global bajar= pose_add ( get_actual_tcp_pose (), bajada_broca)
        $ 3229 "bajar" "breakAfter"
        movel(bajar, a=0.005, v=0.001)
        $ 3230 "subir≔pose_sub(get_actual_tcp_pose(), bajada_broca)"
        global subir= pose_sub ( get_actual_tcp_pose (), bajada_broca)
        $ 3231 "subir" "breakAfter"
        movel(subir, a=0.01, v=0.01)
        $ 3232 "bajada_broca≔pose_sub(bajada_broca, bajada)"
        global bajada_broca= pose_sub (bajada_broca, bajada)
        Loop_21 = Loop_21 + 1
      end
      $ 3233 "Direction: Base Z+"
      global move_thread_flag_3233=0
      thread move_thread_3233():
        enter_critical
        move_thread_flag_3233 = 1
        local towardsPos=calculate_point_to_move_towards(p[0.0,0.0,0.0,0.0,0.0,0.0], [0.0,0.0,1.0], 0.06)
        movel(towardsPos, a=0.035, v=0.03)
        move_thread_flag_3233 = 2
        exit_critical
      end
      move_thread_flag_3233 = 0
      move_thread_han_3233 = run move_thread_3233()
      while (True):
        sleep(1.0E-10)
        if (move_thread_flag_3233 > 1):
          join move_thread_han_3233
          $ 3234 "Until (distance)"
          break
        end
        sync()
      end
      $ 3235 "Set CO[1]=Apagar"
      set_configurable_digital_out(1, False)
      $ 3236 "barreno_actual≔barreno_actual+1"
      global barreno_actual=barreno_actual+1
      $ 3237 "Call Quitar_broca"
      Quitar_broca()
      $ 3238 "Call Poner_broca"
      Poner_broca()
    end
    $ 3239 "CD"
    $ 3240 "'desbaste_inicial'"
    # 'desbaste_inicial'
    $ 3241 "bajada_broca≔p[0,0,-0.008,0,0,0]"
    global bajada_broca=p[0,0,-0.008,0,0,0]
    $ 3242 "barrenos_menos1≔8"
    global barrenos_menos1=8
    $ 3243 "barreno_actual≔0"
    global barreno_actual=0
    $ 3244 "Loop barreno_actual≤barrenos_menos1"
    while (barreno_actual <= barrenos_menos1):
      $ 3245 "Perforacion"
      $ 3246 "MoveL"
      $ 3247 "internos≔interpolate_pose(Linea3_C, Linea3_D, barreno_actual/barrenos_menos1)"
      global internos= interpolate_pose (Linea3_C_p, Linea3_D_p, barreno_actual/barrenos_menos1)
      $ 3248 "internos" "breakAfter"
      movel(internos, a=0.5, v=0.1)
      $ 3249 "'desbaste_inicial'"
      # 'desbaste_inicial'
      $ 3250 "bajada_broca≔p[0,0,-0.008,0,0,0]"
      global bajada_broca=p[0,0,-0.008,0,0,0]
      $ 3251 "bajada≔p[0,0,0.008,0,0,0]"
      global bajada=p[0,0,0.008,0,0,0]
      $ 3252 "Direction: Base Z-"
      global move_thread_flag_3252=0
      thread move_thread_3252():
        enter_critical
        move_thread_flag_3252 = 1
        local towardsPos=calculate_point_to_move_towards(p[0.0,0.0,0.0,0.0,0.0,0.0], [0.0,0.0,-1.0], 0.08)
        movel(towardsPos, a=0.035, v=0.03)
        move_thread_flag_3252 = 2
        exit_critical
      end
      move_thread_flag_3252 = 0
      move_thread_han_3252 = run move_thread_3252()
      while (True):
        sleep(1.0E-10)
        if (move_thread_flag_3252 > 1):
          join move_thread_han_3252
          $ 3253 "Until (distance)"
          break
        end
        sync()
      end
      $ 3254 "Popup: punto contacto alanzdo"
      popup("punto contacto alanzdo", "Mensaje", False, False, blocking=True)
      $ 3255 "Direction: Base Z+"
      global move_thread_flag_3255=0
      thread move_thread_3255():
        enter_critical
        move_thread_flag_3255 = 1
        local towardsPos=calculate_point_to_move_towards(p[0.0,0.0,0.0,0.0,0.0,0.0], [0.0,0.0,1.0], 0.002)
        movel(towardsPos, a=0.005, v=0.003)
        move_thread_flag_3255 = 2
        exit_critical
      end
      move_thread_flag_3255 = 0
      move_thread_han_3255 = run move_thread_3255()
      while (True):
        sleep(1.0E-10)
        if (move_thread_flag_3255 > 1):
          join move_thread_han_3255
          $ 3256 "Until (distance)"
          break
        end
        sync()
      end
      $ 3257 "Wait: 0.3"
      sleep(0.3)
      $ 3258 "Set CO[1]=Encender"
      set_configurable_digital_out(1, True)
      $ 3259 "Wait: 0.3"
      sleep(0.3)
      $ 3260 "Loop 3 times"
      Loop_24 = 0
      while (Loop_24 < 3):
        $ 3261 "bajar≔pose_add(get_actual_tcp_pose(), bajada_broca)"
        global bajar= pose_add ( get_actual_tcp_pose (), bajada_broca)
        $ 3262 "bajar" "breakAfter"
        movel(bajar, a=0.005, v=0.001)
        $ 3263 "subir≔pose_sub(get_actual_tcp_pose(), bajada_broca)"
        global subir= pose_sub ( get_actual_tcp_pose (), bajada_broca)
        $ 3264 "subir" "breakAfter"
        movel(subir, a=0.01, v=0.01)
        $ 3265 "bajada_broca≔pose_sub(bajada_broca, bajada)"
        global bajada_broca= pose_sub (bajada_broca, bajada)
        Loop_24 = Loop_24 + 1
      end
      $ 3266 "Direction: Base Z+"
      global move_thread_flag_3266=0
      thread move_thread_3266():
        enter_critical
        move_thread_flag_3266 = 1
        local towardsPos=calculate_point_to_move_towards(p[0.0,0.0,0.0,0.0,0.0,0.0], [0.0,0.0,1.0], 0.06)
        movel(towardsPos, a=0.035, v=0.03)
        move_thread_flag_3266 = 2
        exit_critical
      end
      move_thread_flag_3266 = 0
      move_thread_han_3266 = run move_thread_3266()
      while (True):
        sleep(1.0E-10)
        if (move_thread_flag_3266 > 1):
          join move_thread_han_3266
          $ 3267 "Until (distance)"
          break
        end
        sync()
      end
      $ 3268 "Set CO[1]=Apagar"
      set_configurable_digital_out(1, False)
      $ 3269 "barreno_actual≔barreno_actual+1"
      global barreno_actual=barreno_actual+1
      $ 3270 "Call Quitar_broca"
      Quitar_broca()
      $ 3271 "Call Poner_broca"
      Poner_broca()
    end
    $ 3272 "EF"
    $ 3273 "'desbaste_inicial'"
    # 'desbaste_inicial'
    $ 3274 "bajada_broca≔p[0,0,-0.008,0,0,0]"
    global bajada_broca=p[0,0,-0.008,0,0,0]
    $ 3275 "barrenos_menos1≔8"
    global barrenos_menos1=8
    $ 3276 "barreno_actual≔0"
    global barreno_actual=0
    $ 3277 "Loop barreno_actual≤barrenos_menos1"
    while (barreno_actual <= barrenos_menos1):
      $ 3278 "Perforacion"
      $ 3279 "MoveL"
      $ 3280 "internos≔interpolate_pose(Linea3_E, Linea3_F, barreno_actual/barrenos_menos1)"
      global internos= interpolate_pose (Linea3_E_p, Linea3_F_p, barreno_actual/barrenos_menos1)
      $ 3281 "internos" "breakAfter"
      movel(internos, a=0.5, v=0.1)
      $ 3282 "'desbaste_inicial'"
      # 'desbaste_inicial'
      $ 3283 "bajada_broca≔p[0,0,-0.008,0,0,0]"
      global bajada_broca=p[0,0,-0.008,0,0,0]
      $ 3284 "bajada≔p[0,0,0.008,0,0,0]"
      global bajada=p[0,0,0.008,0,0,0]
      $ 3285 "Direction: Base Z-"
      global move_thread_flag_3285=0
      thread move_thread_3285():
        enter_critical
        move_thread_flag_3285 = 1
        local towardsPos=calculate_point_to_move_towards(p[0.0,0.0,0.0,0.0,0.0,0.0], [0.0,0.0,-1.0], 0.08)
        movel(towardsPos, a=0.035, v=0.03)
        move_thread_flag_3285 = 2
        exit_critical
      end
      move_thread_flag_3285 = 0
      move_thread_han_3285 = run move_thread_3285()
      while (True):
        sleep(1.0E-10)
        if (move_thread_flag_3285 > 1):
          join move_thread_han_3285
          $ 3286 "Until (distance)"
          break
        end
        sync()
      end
      $ 3287 "Popup: punto contacto alanzdo"
      popup("punto contacto alanzdo", "Mensaje", False, False, blocking=True)
      $ 3288 "Direction: Base Z+"
      global move_thread_flag_3288=0
      thread move_thread_3288():
        enter_critical
        move_thread_flag_3288 = 1
        local towardsPos=calculate_point_to_move_towards(p[0.0,0.0,0.0,0.0,0.0,0.0], [0.0,0.0,1.0], 0.002)
        movel(towardsPos, a=0.005, v=0.003)
        move_thread_flag_3288 = 2
        exit_critical
      end
      move_thread_flag_3288 = 0
      move_thread_han_3288 = run move_thread_3288()
      while (True):
        sleep(1.0E-10)
        if (move_thread_flag_3288 > 1):
          join move_thread_han_3288
          $ 3289 "Until (distance)"
          break
        end
        sync()
      end
      $ 3290 "Wait: 0.3"
      sleep(0.3)
      $ 3291 "Set CO[1]=Encender"
      set_configurable_digital_out(1, True)
      $ 3292 "Wait: 0.3"
      sleep(0.3)
      $ 3293 "Loop 3 times"
      Loop_46 = 0
      while (Loop_46 < 3):
        $ 3294 "bajar≔pose_add(get_actual_tcp_pose(), bajada_broca)"
        global bajar= pose_add ( get_actual_tcp_pose (), bajada_broca)
        $ 3295 "bajar" "breakAfter"
        movel(bajar, a=0.005, v=0.001)
        $ 3296 "subir≔pose_sub(get_actual_tcp_pose(), bajada_broca)"
        global subir= pose_sub ( get_actual_tcp_pose (), bajada_broca)
        $ 3297 "subir" "breakAfter"
        movel(subir, a=0.01, v=0.01)
        $ 3298 "bajada_broca≔pose_sub(bajada_broca, bajada)"
        global bajada_broca= pose_sub (bajada_broca, bajada)
        Loop_46 = Loop_46 + 1
      end
      $ 3299 "Direction: Base Z+"
      global move_thread_flag_3299=0
      thread move_thread_3299():
        enter_critical
        move_thread_flag_3299 = 1
        local towardsPos=calculate_point_to_move_towards(p[0.0,0.0,0.0,0.0,0.0,0.0], [0.0,0.0,1.0], 0.06)
        movel(towardsPos, a=0.035, v=0.03)
        move_thread_flag_3299 = 2
        exit_critical
      end
      move_thread_flag_3299 = 0
      move_thread_han_3299 = run move_thread_3299()
      while (True):
        sleep(1.0E-10)
        if (move_thread_flag_3299 > 1):
          join move_thread_han_3299
          $ 3300 "Until (distance)"
          break
        end
        sync()
      end
      $ 3301 "Set CO[1]=Apagar"
      set_configurable_digital_out(1, False)
      $ 3302 "barreno_actual≔barreno_actual+1"
      global barreno_actual=barreno_actual+1
      $ 3303 "Call Quitar_broca"
      Quitar_broca()
      $ 3304 "Call Poner_broca"
      Poner_broca()
    end
    $ 3305 "Popup: Linea3 con chica Terminada!"
    popup("Linea3 con chica Terminada!", "Mensaje", False, False, blocking=True)
    $ 3306 "Linea4"
    $ 3307 "Marcar_puntos"
    $ 3308 "MoveL"
    $ 3309 "Home3" "breakAfter"
    movel(Home3_p, a=0.5, v=0.1)
    $ 3310 "Linea4_A" "breakAfter"
    movel(Linea4_A_p, a=0.5, v=0.1)
    $ 3311 "Linea4_B" "breakAfter"
    movel(Linea4_B_p, a=0.5, v=0.1)
    $ 3312 "Linea4_C" "breakAfter"
    movel(Linea4_C_p, a=0.5, v=0.1)
    $ 3313 "Linea4_D" "breakAfter"
    movel(Linea4_D_p, a=0.5, v=0.1)
    $ 3314 "Linea4_E" "breakAfter"
    movel(Linea4_E_p, a=0.5, v=0.1)
    $ 3315 "Linea4_F" "breakAfter"
    movel(Linea4_F_p, a=0.5, v=0.1)
    $ 3316 "AB"
    $ 3317 "'desbaste_inicial'"
    # 'desbaste_inicial'
    $ 3318 "bajada_broca≔p[0,0,-0.008,0,0,0]"
    global bajada_broca=p[0,0,-0.008,0,0,0]
    $ 3319 "barrenos_menos1≔8"
    global barrenos_menos1=8
    $ 3320 "barreno_actual≔0"
    global barreno_actual=0
    $ 3321 "Loop barreno_actual≤barrenos_menos1"
    while (barreno_actual <= barrenos_menos1):
      $ 3322 "Perforacion"
      $ 3323 "MoveL"
      $ 3324 "internos≔interpolate_pose(Linea4_A, Linea4_B, barreno_actual/barrenos_menos1)"
      global internos= interpolate_pose (Linea4_A_p, Linea4_B_p, barreno_actual/barrenos_menos1)
      $ 3325 "internos" "breakAfter"
      movel(internos, a=0.5, v=0.1)
      $ 3326 "'desbaste_inicial'"
      # 'desbaste_inicial'
      $ 3327 "bajada_broca≔p[0,0,-0.008,0,0,0]"
      global bajada_broca=p[0,0,-0.008,0,0,0]
      $ 3328 "bajada≔p[0,0,0.008,0,0,0]"
      global bajada=p[0,0,0.008,0,0,0]
      $ 3329 "Direction: Base Z-"
      global move_thread_flag_3329=0
      thread move_thread_3329():
        enter_critical
        move_thread_flag_3329 = 1
        local towardsPos=calculate_point_to_move_towards(p[0.0,0.0,0.0,0.0,0.0,0.0], [0.0,0.0,-1.0], 0.08)
        movel(towardsPos, a=0.035, v=0.03)
        move_thread_flag_3329 = 2
        exit_critical
      end
      move_thread_flag_3329 = 0
      move_thread_han_3329 = run move_thread_3329()
      while (True):
        sleep(1.0E-10)
        if (move_thread_flag_3329 > 1):
          join move_thread_han_3329
          $ 3330 "Until (distance)"
          break
        end
        sync()
      end
      $ 3331 "Popup: punto contacto alanzdo"
      popup("punto contacto alanzdo", "Mensaje", False, False, blocking=True)
      $ 3332 "Direction: Base Z+"
      global move_thread_flag_3332=0
      thread move_thread_3332():
        enter_critical
        move_thread_flag_3332 = 1
        local towardsPos=calculate_point_to_move_towards(p[0.0,0.0,0.0,0.0,0.0,0.0], [0.0,0.0,1.0], 0.002)
        movel(towardsPos, a=0.005, v=0.003)
        move_thread_flag_3332 = 2
        exit_critical
      end
      move_thread_flag_3332 = 0
      move_thread_han_3332 = run move_thread_3332()
      while (True):
        sleep(1.0E-10)
        if (move_thread_flag_3332 > 1):
          join move_thread_han_3332
          $ 3333 "Until (distance)"
          break
        end
        sync()
      end
      $ 3334 "Wait: 0.3"
      sleep(0.3)
      $ 3335 "Set CO[1]=Encender"
      set_configurable_digital_out(1, True)
      $ 3336 "Wait: 0.3"
      sleep(0.3)
      $ 3337 "Loop 3 times"
      Loop_50 = 0
      while (Loop_50 < 3):
        $ 3338 "bajar≔pose_add(get_actual_tcp_pose(), bajada_broca)"
        global bajar= pose_add ( get_actual_tcp_pose (), bajada_broca)
        $ 3339 "bajar" "breakAfter"
        movel(bajar, a=0.005, v=0.001)
        $ 3340 "subir≔pose_sub(get_actual_tcp_pose(), bajada_broca)"
        global subir= pose_sub ( get_actual_tcp_pose (), bajada_broca)
        $ 3341 "subir" "breakAfter"
        movel(subir, a=0.01, v=0.01)
        $ 3342 "bajada_broca≔pose_sub(bajada_broca, bajada)"
        global bajada_broca= pose_sub (bajada_broca, bajada)
        Loop_50 = Loop_50 + 1
      end
      $ 3343 "Direction: Base Z+"
      global move_thread_flag_3343=0
      thread move_thread_3343():
        enter_critical
        move_thread_flag_3343 = 1
        local towardsPos=calculate_point_to_move_towards(p[0.0,0.0,0.0,0.0,0.0,0.0], [0.0,0.0,1.0], 0.06)
        movel(towardsPos, a=0.035, v=0.03)
        move_thread_flag_3343 = 2
        exit_critical
      end
      move_thread_flag_3343 = 0
      move_thread_han_3343 = run move_thread_3343()
      while (True):
        sleep(1.0E-10)
        if (move_thread_flag_3343 > 1):
          join move_thread_han_3343
          $ 3344 "Until (distance)"
          break
        end
        sync()
      end
      $ 3345 "Set CO[1]=Apagar"
      set_configurable_digital_out(1, False)
      $ 3346 "barreno_actual≔barreno_actual+1"
      global barreno_actual=barreno_actual+1
      $ 3347 "Call Quitar_broca"
      Quitar_broca()
      $ 3348 "Call Poner_broca"
      Poner_broca()
    end
    $ 3349 "CD"
    $ 3350 "'desbaste_inicial'"
    # 'desbaste_inicial'
    $ 3351 "bajada_broca≔p[0,0,-0.008,0,0,0]"
    global bajada_broca=p[0,0,-0.008,0,0,0]
    $ 3352 "barrenos_menos1≔8"
    global barrenos_menos1=8
    $ 3353 "barreno_actual≔0"
    global barreno_actual=0
    $ 3354 "Loop barreno_actual≤barrenos_menos1"
    while (barreno_actual <= barrenos_menos1):
      $ 3355 "Perforacion"
      $ 3356 "MoveL"
      $ 3357 "internos≔interpolate_pose(Linea4_C, Linea4_D, barreno_actual/barrenos_menos1)"
      global internos= interpolate_pose (Linea4_C_p, Linea4_D_p, barreno_actual/barrenos_menos1)
      $ 3358 "internos" "breakAfter"
      movel(internos, a=0.5, v=0.1)
      $ 3359 "'desbaste_inicial'"
      # 'desbaste_inicial'
      $ 3360 "bajada_broca≔p[0,0,-0.008,0,0,0]"
      global bajada_broca=p[0,0,-0.008,0,0,0]
      $ 3361 "bajada≔p[0,0,0.008,0,0,0]"
      global bajada=p[0,0,0.008,0,0,0]
      $ 3362 "Direction: Base Z-"
      global move_thread_flag_3362=0
      thread move_thread_3362():
        enter_critical
        move_thread_flag_3362 = 1
        local towardsPos=calculate_point_to_move_towards(p[0.0,0.0,0.0,0.0,0.0,0.0], [0.0,0.0,-1.0], 0.08)
        movel(towardsPos, a=0.035, v=0.03)
        move_thread_flag_3362 = 2
        exit_critical
      end
      move_thread_flag_3362 = 0
      move_thread_han_3362 = run move_thread_3362()
      while (True):
        sleep(1.0E-10)
        if (move_thread_flag_3362 > 1):
          join move_thread_han_3362
          $ 3363 "Until (distance)"
          break
        end
        sync()
      end
      $ 3364 "Popup: punto contacto alanzdo"
      popup("punto contacto alanzdo", "Mensaje", False, False, blocking=True)
      $ 3365 "Direction: Base Z+"
      global move_thread_flag_3365=0
      thread move_thread_3365():
        enter_critical
        move_thread_flag_3365 = 1
        local towardsPos=calculate_point_to_move_towards(p[0.0,0.0,0.0,0.0,0.0,0.0], [0.0,0.0,1.0], 0.002)
        movel(towardsPos, a=0.005, v=0.003)
        move_thread_flag_3365 = 2
        exit_critical
      end
      move_thread_flag_3365 = 0
      move_thread_han_3365 = run move_thread_3365()
      while (True):
        sleep(1.0E-10)
        if (move_thread_flag_3365 > 1):
          join move_thread_han_3365
          $ 3366 "Until (distance)"
          break
        end
        sync()
      end
      $ 3367 "Wait: 0.3"
      sleep(0.3)
      $ 3368 "Set CO[1]=Encender"
      set_configurable_digital_out(1, True)
      $ 3369 "Wait: 0.3"
      sleep(0.3)
      $ 3370 "Loop 3 times"
      Loop_53 = 0
      while (Loop_53 < 3):
        $ 3371 "bajar≔pose_add(get_actual_tcp_pose(), bajada_broca)"
        global bajar= pose_add ( get_actual_tcp_pose (), bajada_broca)
        $ 3372 "bajar" "breakAfter"
        movel(bajar, a=0.005, v=0.001)
        $ 3373 "subir≔pose_sub(get_actual_tcp_pose(), bajada_broca)"
        global subir= pose_sub ( get_actual_tcp_pose (), bajada_broca)
        $ 3374 "subir" "breakAfter"
        movel(subir, a=0.01, v=0.01)
        $ 3375 "bajada_broca≔pose_sub(bajada_broca, bajada)"
        global bajada_broca= pose_sub (bajada_broca, bajada)
        Loop_53 = Loop_53 + 1
      end
      $ 3376 "Direction: Base Z+"
      global move_thread_flag_3376=0
      thread move_thread_3376():
        enter_critical
        move_thread_flag_3376 = 1
        local towardsPos=calculate_point_to_move_towards(p[0.0,0.0,0.0,0.0,0.0,0.0], [0.0,0.0,1.0], 0.06)
        movel(towardsPos, a=0.035, v=0.03)
        move_thread_flag_3376 = 2
        exit_critical
      end
      move_thread_flag_3376 = 0
      move_thread_han_3376 = run move_thread_3376()
      while (True):
        sleep(1.0E-10)
        if (move_thread_flag_3376 > 1):
          join move_thread_han_3376
          $ 3377 "Until (distance)"
          break
        end
        sync()
      end
      $ 3378 "Set CO[1]=Apagar"
      set_configurable_digital_out(1, False)
      $ 3379 "barreno_actual≔barreno_actual+1"
      global barreno_actual=barreno_actual+1
      $ 3380 "Call Quitar_broca"
      Quitar_broca()
      $ 3381 "Call Poner_broca"
      Poner_broca()
    end
    $ 3382 "EF"
    $ 3383 "'desbaste_inicial'"
    # 'desbaste_inicial'
    $ 3384 "bajada_broca≔p[0,0,-0.008,0,0,0]"
    global bajada_broca=p[0,0,-0.008,0,0,0]
    $ 3385 "barrenos_menos1≔8"
    global barrenos_menos1=8
    $ 3386 "barreno_actual≔0"
    global barreno_actual=0
    $ 3387 "Loop barreno_actual≤barrenos_menos1"
    while (barreno_actual <= barrenos_menos1):
      $ 3388 "Perforacion"
      $ 3389 "MoveL"
      $ 3390 "internos≔interpolate_pose(Linea4_E, Linea4_F, barreno_actual/barrenos_menos1)"
      global internos= interpolate_pose (Linea4_E_p, Linea4_F_p, barreno_actual/barrenos_menos1)
      $ 3391 "internos" "breakAfter"
      movel(internos, a=0.5, v=0.1)
